KUKA KRL program: MyProgram_182().src

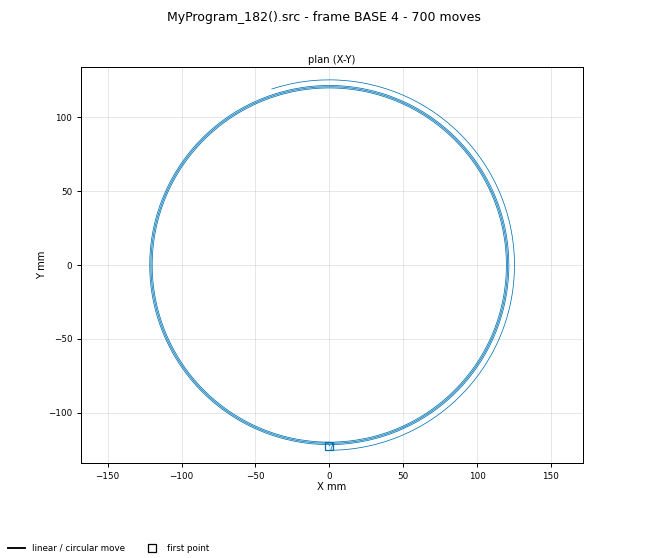
[picture p0: tool path of MyProgram_182().src in frame BASE 4, 700 of 700 moves have a stored position in this frame; points joined in program order, loops and branches not executed]
&ACCESS RVP
&REL 1
&PARAM TEMPLATE = C:\KRC\Roboter\Template\vorgabe
&PARAM EDITMASK = *
DEF MyProgram_182()
; ---- Setting reference (Base) ----
$BASE = BASE_DATA[4]

; --------------------------
; ---- Setting tool (TCP) ----
$TOOL = TOOL_DATA[3]
; --------------------------

$VEL.CP = VEL_APROX_PRINT
Startdeposition()
$VEL.CP = VEL_PRINT
LIN {X -0.1714,Y -122.3614,Z 133,A -93.0303,B 24.9608,C -1.4469,E1 25.0014,E2 179.2424} C_DIS
Enddeposition()
LIN {X 0.8695,Y -121.5175,Z 133,A -93.1539,B 24.9616,C -1.4326,E1 25.001,E2 179.3998} C_DIS
Startdeposition()
$VEL.CP = VEL_PRINT
LIN {X -1.6199,Y -121.5128,Z 133,A -95.084,B 24.9634,C -1.3971,E1 24.9954,E2 181.4142} C_DIS
LIN {X -5.9089,Y -121.3798,Z 133,A -96.2452,B 24.9613,C -1.437,E1 24.9924,E2 182.4809} C_DIS
LIN {X -12.044,Y -120.9259,Z 133,A -99.4115,B 24.962,C -1.4246,E1 24.9835,E2 185.6781} C_DIS
LIN {X -17.4797,Y -120.2602,Z 133,A -101.7782,B 24.9614,C -1.435,E1 24.977,E2 188.0216} C_DIS
LIN {X -21.0401,Y -119.6879,Z 133,A -103.7397,B 24.962,C -1.4234,E1 24.9715,E2 190.0125} C_DIS
LIN {X -24.264,Y -119.0756,Z 133,A -105.5719,B 24.9627,C -1.411,E1 24.9664,E2 191.8764} C_DIS
LIN {X -29.5809,Y -117.8675,Z 133,A -107.8497,B 24.9619,C -1.4258,E1 24.9603,E2 194.1221} C_DIS
LIN {X -32.4256,Y -117.1176,Z 133,A -109.326,B 24.9621,C -1.4225,E1 24.9563,E2 195.6083} C_DIS
LIN {X -36.1039,Y -116.0375,Z 133,A -111.1589,B 24.9621,C -1.4227,E1 24.9514,E2 197.444} C_DIS
LIN {X -40.6433,Y -114.5267,Z 133,A -113.43,B 24.9621,C -1.4239,E1 24.9454,E2 199.7166} C_DIS
LIN {X -44.0347,Y -113.2641,Z 133,A -115.0276,B 24.9617,C -1.4305,E1 24.9412,E2 201.3019} C_DIS
LIN {X -49.4851,Y -110.9909,Z 133,A -117.8563,B 24.9617,C -1.4314,E1 24.934,E2 204.1348} C_DIS
LIN {X -52.5926,Y -109.5528,Z 133,A -119.7843,B 24.9623,C -1.4192,E1 24.929,E2 206.0968} C_DIS
LIN {X -55.6549,Y -108.031,Z 133,A -121.1723,B 24.9616,C -1.4313,E1 24.9256,E2 207.4598} C_DIS
LIN {X -59.6628,Y -105.8704,Z 133,A -123.3001,B 24.9614,C -1.4352,E1 24.9204,E2 209.5846} C_DIS
LIN {X -62.5934,Y -104.165,Z 133,A -125.1136,B 24.9618,C -1.4279,E1 24.916,E2 211.4209} C_DIS
LIN {X -66.9605,Y -101.4123,Z 133,A -127.3139,B 24.961,C -1.4422,E1 24.9109,E2 213.5943} C_DIS
LIN {X -72.1767,Y -97.7684,Z 133,A -130.3221,B 24.9608,C -1.4469,E1 24.9041,E2 216.6016} C_DIS
LIN {X -75.3691,Y -95.3299,Z 133,A -132.2793,B 24.9608,C -1.4476,E1 24.8998,E2 218.5644} C_DIS
LIN {X -78.4994,Y -92.7685,Z 133,A -134.1769,B 24.9605,C -1.4517,E1 24.8957,E2 220.4595} C_DIS
LIN {X -81.6362,Y -90.0204,Z 133,A -135.8524,B 24.9596,C -1.4685,E1 24.8923,E2 222.1017} C_DIS
LIN {X -84.8955,Y -86.9542,Z 133,A -138.4312,B 24.9605,C -1.4522,E1 24.887,E2 224.7299} C_DIS
LIN {X -88.5295,Y -83.2516,Z 133,A -140.5025,B 24.9593,C -1.4741,E1 24.883,E2 226.7581} C_DIS
LIN {X -90.7073,Y -80.8729,Z 133,A -142.282,B 24.9597,C -1.4661,E1 24.8796,E2 228.5643} C_DIS
LIN {X -93.9091,Y -77.1324,Z 133,A -144.7365,B 24.9597,C -1.4658,E1 24.8752,E2 231.0309} C_DIS
LIN {X -96.8725,Y -73.375,Z 133,A -146.936,B 24.9593,C -1.4738,E1 24.8715,E2 233.2217} C_DIS
LIN {X -99.5155,Y -69.7483,Z 133,A -148.943,B 24.9587,C -1.4839,E1 24.8682,E2 235.2145} C_DIS
LIN {X -101.2493,Y -67.2069,Z 133,A -150.5671,B 24.959,C -1.4802,E1 24.8657,E2 236.8557} C_DIS
LIN {X -103.6846,Y -63.3844,Z 133,A -152.5823,B 24.9583,C -1.4911,E1 24.8627,E2 238.8551} C_DIS
LIN {X -105.425,Y -60.4464,Z 133,A -154.7129,B 24.9593,C -1.4731,E1 24.8597,E2 241.0398} C_DIS
LIN {X -107.529,Y -56.6154,Z 133,A -156.1389,B 24.9575,C -1.5062,E1 24.8579,E2 242.3945} C_DIS
LIN {X -109.0325,Y -53.6618,Z 133,A -157.753,B 24.9574,C -1.5083,E1 24.8559,E2 244.0121} C_DIS
LIN {X -110.2041,Y -51.2135,Z 133,A -159.1619,B 24.9574,C -1.5064,E1 24.8542,E2 245.4333} C_DIS
LIN {X -112.0151,Y -47.1208,Z 133,A -161.1145,B 24.9568,C -1.5194,E1 24.852,E2 247.3658} C_DIS
LIN {X -113.0996,Y -44.4581,Z 133,A -162.6444,B 24.957,C -1.5159,E1 24.8504,E2 248.9126} C_DIS
LIN {X -114.5797,Y -40.4958,Z 133,A -165.1319,B 24.9578,C -1.5007,E1 24.8481,E2 251.4502} C_DIS
LIN {X -115.9774,Y -36.2992,Z 133,A -166.7405,B 24.9563,C -1.5274,E1 24.8467,E2 253.0044} C_DIS
LIN {X -117.0095,Y -32.8111,Z 133,A -168.3362,B 24.9557,C -1.5379,E1 24.8455,E2 254.5845} C_DIS
LIN {X -117.8307,Y -29.726,Z 133,A -169.9109,B 24.9556,C -1.5396,E1 24.8444,E2 256.1642} C_DIS
LIN {X -118.7261,Y -25.9215,Z 133,A -171.7761,B 24.9553,C -1.5444,E1 24.8432,E2 258.0289} C_DIS
LIN {X -119.4847,Y -22.1777,Z 133,A -173.7085,B 24.9553,C -1.5444,E1 24.8422,E2 259.9726} C_DIS
LIN {X -120.082,Y -18.6588,Z 133,A -175.2045,B 24.9545,C -1.5579,E1 24.8416,E2 261.4455} C_DIS
LIN {X -120.5511,Y -15.3426,Z 133,A -177.0022,B 24.9548,C -1.5536,E1 24.8409,E2 263.2642} C_DIS
LIN {X -121.1464,Y -9.5742,Z 133,A -179.7063,B 24.9542,C -1.5637,E1 24.8402,E2 265.9603} C_DIS
LIN {X -121.3814,Y -5.8756,Z 133,A 178.598,B 24.9537,C -1.5716,E1 24.8399,E2 267.6474} C_DIS
LIN {X -121.5254,Y 0.0221,Z 133,A 175.7482,B 24.9534,C -1.5778,E1 24.8398,E2 270.4998} C_DIS
LIN {X -121.3885,Y 5.7327,Z 133,A 173.2315,B 24.9524,C -1.5941,E1 24.84,E2 272.9926} C_DIS
LIN {X -121.191,Y 8.9707,Z 133,A 171.3253,B 24.953,C -1.5832,E1 24.8404,E2 274.9364} C_DIS
LIN {X -120.7228,Y 13.9263,Z 133,A 169.1754,B 24.9521,C -1.5992,E1 24.841,E2 277.061} C_DIS
LIN {X -120.2359,Y 17.6498,Z 133,A 167.4666,B 24.9516,C -1.6076,E1 24.8416,E2 278.7599} C_DIS
LIN {X -119.6712,Y 21.1333,Z 133,A 165.9207,B 24.9509,C -1.6181,E1 24.8423,E2 280.2901} C_DIS
LIN {X -119.212,Y 23.5938,Z 133,A 164.3598,B 24.9517,C -1.6057,E1 24.8432,E2 281.8898} C_DIS
LIN {X -118.2189,Y 28.1465,Z 133,A 162.2925,B 24.9509,C -1.6183,E1 24.8445,E2 283.9391} C_DIS
LIN {X -117.2416,Y 31.9811,Z 133,A 160.3797,B 24.9507,C -1.6223,E1 24.8458,E2 285.8536} C_DIS
LIN {X -116.311,Y 35.2093,Z 133,A 158.6706,B 24.9507,C -1.622,E1 24.8472,E2 287.5731} C_DIS
LIN {X -114.606,Y 40.4198,Z 133,A 156.1475,B 24.95,C -1.6328,E1 24.8495,E2 290.0849} C_DIS
LIN {X -113.2622,Y 44.0395,Z 133,A 154.6517,B 24.9488,C -1.6524,E1 24.8509,E2 291.5424} C_DIS
LIN {X -111.9631,Y 47.2453,Z 133,A 152.7073,B 24.9494,C -1.6441,E1 24.853,E2 293.5175} C_DIS
LIN {X -110.3469,Y 50.9041,Z 133,A 150.9642,B 24.9486,C -1.656,E1 24.855,E2 295.2419} C_DIS
LIN {X -109.2384,Y 53.245,Z 133,A 149.0187,B 24.9503,C -1.6289,E1 24.8575,E2 297.2624} C_DIS
LIN {X -107.0191,Y 57.5774,Z 133,A 146.7211,B 24.9499,C -1.6356,E1 24.8605,E2 299.5562} C_DIS
LIN {X -104.6811,Y 61.7255,Z 133,A 145.3326,B 24.9472,C -1.6786,E1 24.8623,E2 300.8493} C_DIS
LIN {X -100.2308,Y 68.7165,Z 133,A 141.1386,B 24.9472,C -1.6774,E1 24.8687,E2 305.0674} C_DIS
LIN {X -97.9703,Y 71.9019,Z 133,A 139.3158,B 24.9469,C -1.6833,E1 24.8716,E2 306.8851} C_DIS
LIN {X -95.4946,Y 75.1596,Z 133,A 137.3071,B 24.9468,C -1.6851,E1 24.8751,E2 308.8989} C_DIS
LIN {X -92.8236,Y 78.4345,Z 133,A 135.3193,B 24.9464,C -1.6906,E1 24.8786,E2 310.8829} C_DIS
LIN {X -90.3001,Y 81.3277,Z 133,A 133.4255,B 24.9464,C -1.6916,E1 24.8821,E2 312.7827} C_DIS
LIN {X -87.1093,Y 84.7363,Z 133,A 131.2611,B 24.9459,C -1.6988,E1 24.8863,E2 314.9396} C_DIS
LIN {X -84.2652,Y 87.5645,Z 133,A 129.3791,B 24.9456,C -1.7037,E1 24.89,E2 316.8175} C_DIS
LIN {X -81.1545,Y 90.4552,Z 133,A 127.342,B 24.9454,C -1.7069,E1 24.8942,E2 318.8552} C_DIS
LIN {X -77.9713,Y 93.2126,Z 133,A 125.4465,B 24.9449,C -1.7154,E1 24.8982,E2 320.738} C_DIS
LIN {X -74.8032,Y 95.7746,Z 133,A 123.3839,B 24.9449,C -1.7134,E1 24.9028,E2 322.813} C_DIS
LIN {X -71.0844,Y 98.5665,Z 133,A 121.1715,B 24.9447,C -1.7171,E1 24.9077,E2 325.0243} C_DIS
LIN {X -67.5256,Y 101.0364,Z 133,A 119.4573,B 24.9435,C -1.7356,E1 24.9116,E2 326.7003} C_DIS
LIN {X -64.1253,Y 103.2284,Z 133,A 117.0152,B 24.9448,C -1.7159,E1 24.9175,E2 329.1971} C_DIS
LIN {X -61.3323,Y 104.9117,Z 133,A 115.7211,B 24.944,C -1.7293,E1 24.9205,E2 330.4632} C_DIS
LIN {X -57.7529,Y 106.9251,Z 133,A 113.5487,B 24.9444,C -1.7223,E1 24.9259,E2 332.6585} C_DIS
LIN {X -53.5846,Y 109.0707,Z 133,A 111.6337,B 24.9433,C -1.739,E1 24.9306,E2 334.5389} C_DIS
LIN {X -49.7713,Y 110.8628,Z 133,A 109.6684,B 24.9431,C -1.743,E1 24.9356,E2 336.4995} C_DIS
LIN {X -47.024,Y 112.0556,Z 133,A 108.269,B 24.9429,C -1.7457,E1 24.9392,E2 337.8959} C_DIS
LIN {X -41.3309,Y 114.2785,Z 133,A 105.3623,B 24.9427,C -1.7484,E1 24.9468,E2 340.8022} C_DIS
LIN {X -38.0593,Y 115.4093,Z 133,A 103.6121,B 24.9429,C -1.7452,E1 24.9514,E2 342.5634} C_DIS
LIN {X -33.9229,Y 116.6918,Z 133,A 101.5952,B 24.9427,C -1.7486,E1 24.9568,E2 344.5756} C_DIS
LIN {X -30.0844,Y 117.7399,Z 133,A 99.7639,B 24.9424,C -1.7525,E1 24.9617,E2 346.4004} C_DIS
LIN {X -27.4403,Y 118.3855,Z 133,A 98.1282,B 24.9434,C -1.7379,E1 24.9663,E2 348.0729} C_DIS
LIN {X -24.2011,Y 119.0884,Z 133,A 97.0595,B 24.9418,C -1.7614,E1 24.969,E2 349.087} C_DIS
LIN {X -18.4586,Y 120.113,Z 133,A 94.1674,B 24.9421,C -1.7571,E1 24.977,E2 351.9923} C_DIS
LIN {X -15.4534,Y 120.5366,Z 133,A 91.9287,B 24.9444,C -1.7217,E1 24.9835,E2 354.3165} C_DIS
LIN {X -9.9847,Y 121.1119,Z 133,A 90.4873,B 24.941,C -1.7749,E1 24.9871,E2 355.6325} C_DIS
LIN {X -4.1146,Y 121.4544,Z 133,A 87.4557,B 24.9417,C -1.764,E1 24.9957,E2 358.6908} C_DIS
LIN {X 2.7806,Y 121.4924,Z 133,A 83.7604,B 24.943,C -1.7443,E1 25.0061,E2 362.4325} C_DIS
LIN {X 6.1114,Y 121.3697,Z 133,A 82.3946,B 24.9424,C -1.7538,E1 25.0098,E2 363.7754} C_DIS
LIN {X 9.304,Y 121.1666,Z 133,A 80.4497,B 24.9437,C -1.7338,E1 25.0154,E2 365.7668} C_DIS
LIN {X 13.7722,Y 120.7407,Z 133,A 78.9161,B 24.9419,C -1.7601,E1 25.0195,E2 367.237} C_DIS
LIN {X 17.8606,Y 120.2057,Z 133,A 76.8319,B 24.9424,C -1.7531,E1 25.0253,E2 369.336} C_DIS
LIN {X 21.3951,Y 119.6246,Z 133,A 75.0487,B 24.9427,C -1.7482,E1 25.0302,E2 371.129} C_DIS
LIN {X 26.4333,Y 118.6147,Z 133,A 72.8052,B 24.9423,C -1.7552,E1 25.0363,E2 373.3528} C_DIS
LIN {X 30.0915,Y 117.7381,Z 133,A 71.1132,B 24.9421,C -1.758,E1 25.0408,E2 375.0358} C_DIS
LIN {X 33.5438,Y 116.8029,Z 133,A 69.4281,B 24.9421,C -1.7569,E1 25.0454,E2 376.7208} C_DIS
LIN {X 37.679,Y 115.5357,Z 133,A 67.2523,B 24.9427,C -1.7489,E1 25.0512,E2 378.9115} C_DIS
LIN {X 40.9856,Y 114.4031,Z 133,A 65.7299,B 24.9424,C -1.7533,E1 25.0552,E2 380.4204} C_DIS
LIN {X 47.3838,Y 111.9053,Z 133,A 62.4044,B 24.9429,C -1.7458,E1 25.0638,E2 383.7561} C_DIS
LIN {X 52.9272,Y 109.3927,Z 133,A 59.5132,B 24.9432,C -1.7414,E1 25.0712,E2 386.6505} C_DIS
LIN {X 56.3187,Y 107.6851,Z 133,A 57.82,B 24.943,C -1.7436,E1 25.0754,E2 388.3338} C_DIS
LIN {X 59.7529,Y 105.8199,Z 133,A 55.319,B 24.9452,C -1.7099,E1 25.0816,E2 390.907} C_DIS
LIN {X 64.0474,Y 103.2768,Z 133,A 53.7251,B 24.9431,C -1.7422,E1 25.0852,E2 392.4197} C_DIS
LIN {X 69.0589,Y 99.9957,Z 133,A 50.7198,B 24.944,C -1.7289,E1 25.0923,E2 395.4464} C_DIS
LIN {X 72.9607,Y 97.1859,Z 133,A 48.6037,B 24.9438,C -1.7321,E1 25.097,E2 397.5474} C_DIS
LIN {X 75.8072,Y 94.9809,Z 133,A 46.8061,B 24.9443,C -1.7241,E1 25.101,E2 399.3572} C_DIS
LIN {X 79.2112,Y 92.1619,Z 133,A 44.7655,B 24.9444,C -1.7221,E1 25.1053,E2 401.3946} C_DIS
LIN {X 82.2523,Y 89.4574,Z 133,A 43.1469,B 24.9437,C -1.7327,E1 25.1086,E2 402.9817} C_DIS
LIN {X 85.4415,Y 86.4173,Z 133,A 40.7559,B 24.945,C -1.7131,E1 25.1135,E2 405.4091} C_DIS
LIN {X 88.7384,Y 83.0292,Z 133,A 38.49,B 24.9454,C -1.7063,E1 25.1179,E2 407.6811} C_DIS
LIN {X 91.8422,Y 79.5817,Z 133,A 36.4182,B 24.9454,C -1.7068,E1 25.1217,E2 409.7424} C_DIS
LIN {X 95.331,Y 75.3678,Z 133,A 33.7885,B 24.946,C -1.6982,E1 25.1263,E2 412.3805} C_DIS
LIN {X 97.7085,Y 72.2582,Z 133,A 31.9897,B 24.9461,C -1.6958,E1 25.1294,E2 414.1761} C_DIS
LIN {X 101.2183,Y 67.2533,Z 133,A 29.0556,B 24.9467,C -1.6859,E1 25.134,E2 417.1193} C_DIS
LIN {X 103.1728,Y 64.215,Z 133,A 27.6255,B 24.9462,C -1.6947,E1 25.1361,E2 418.5213} C_DIS
LIN {X 105.044,Y 61.1053,Z 133,A 25.7489,B 24.947,C -1.6819,E1 25.1388,E2 420.4184} C_DIS
LIN {X 107.0074,Y 57.5991,Z 133,A 23.8134,B 24.9474,C -1.6747,E1 25.1414,E2 422.361} C_DIS
LIN {X 109.006,Y 53.7155,Z 133,A 21.2767,B 24.9493,C -1.6455,E1 25.1447,E2 424.9529} C_DIS
LIN {X 110.9245,Y 49.6335,Z 133,A 19.6987,B 24.948,C -1.6662,E1 25.1464,E2 426.4735} C_DIS
LIN {X 112.5458,Y 45.8395,Z 133,A 17.6274,B 24.9487,C -1.6543,E1 25.1487,E2 428.5616} C_DIS
LIN {X 114.2892,Y 41.3014,Z 133,A 15.5706,B 24.9484,C -1.659,E1 25.1506,E2 430.5957} C_DIS
LIN {X 115.4115,Y 38.0527,Z 133,A 13.8382,B 24.9491,C -1.6486,E1 25.1522,E2 432.343} C_DIS
LIN {X 116.909,Y 33.1693,Z 133,A 11.4999,B 24.9493,C -1.6446,E1 25.1541,E2 434.6773} C_DIS
LIN {X 117.9396,Y 29.2965,Z 133,A 9.2966,B 24.9506,C -1.6232,E1 25.1556,E2 436.9183} C_DIS
LIN {X 118.7103,Y 25.9949,Z 133,A 7.7401,B 24.9508,C -1.6202,E1 25.1565,E2 438.4728} C_DIS
LIN {X 119.3724,Y 22.7623,Z 133,A 6.0818,B 24.9514,C -1.6102,E1 25.1574,E2 440.1449} C_DIS
LIN {X 120.032,Y 18.9807,Z 133,A 3.7513,B 24.9533,C -1.5789,E1 25.1584,E2 442.5357} C_DIS
LIN {X 120.8602,Y 12.6811,Z 133,A 1.024,B 24.9531,C -1.5823,E1 25.1592,E2 445.2387} C_DIS
LIN {X 121.2876,Y 7.5595,Z 133,A -0.6208,B 24.9513,C -1.6129,E1 25.1595,E2 446.8016} C_DIS
LIN {X 121.5233,Y 0.4226,Z 133,A -3.7776,B 24.9513,C -1.6123,E1 25.1598,E2 449.941} C_DIS
LIN {X 121.5038,Y -2.1482,Z 133,A -5.3004,B 24.9525,C -1.5928,E1 25.1598,E2 451.5006} C_DIS
LIN {X 121.3612,Y -6.2818,Z 133,A -7.1686,B 24.9526,C -1.5905,E1 25.1595,E2 453.3633} C_DIS
LIN {X 121.0842,Y -10.3146,Z 133,A -8.9077,B 24.9525,C -1.5926,E1 25.1592,E2 455.0872} C_DIS
LIN {X 120.1422,Y -18.2707,Z 133,A -12.5694,B 24.9529,C -1.5859,E1 25.1579,E2 458.743} C_DIS
LIN {X 119.0748,Y -24.2677,Z 133,A -15.5726,B 24.9538,C -1.5699,E1 25.1564,E2 461.7664} C_DIS
LIN {X 117.9952,Y -29.0716,Z 133,A -18.0282,B 24.9547,C -1.5556,E1 25.1548,E2 464.2413} C_DIS
LIN {X 117.0701,Y -32.595,Z 133,A -19.6657,B 24.9547,C -1.5541,E1 25.1536,E2 465.8729} C_DIS
LIN {X 114.9989,Y -39.2852,Z 133,A -22.999,B 24.9555,C -1.542,E1 25.1508,E2 469.216} C_DIS
LIN {X 113.7527,Y -42.7553,Z 133,A -24.6508,B 24.9555,C -1.5408,E1 25.1492,E2 470.8612} C_DIS
LIN {X 112.8471,Y -45.0941,Z 133,A -26.4568,B 24.9575,C -1.5062,E1 25.1473,E2 472.7388} C_DIS
LIN {X 111.0301,Y -49.3975,Z 133,A -28.0517,B 24.9562,C -1.5294,E1 25.1456,E2 474.2703} C_DIS
LIN {X 109.6975,Y -52.2901,Z 133,A -29.4513,B 24.9562,C -1.5299,E1 25.1439,E2 475.6612} C_DIS
LIN {X 108.5654,Y -54.6031,Z 133,A -31.582,B 24.9589,C -1.481,E1 25.1411,E2 477.8959} C_DIS
LIN {X 105.7915,Y -59.8034,Z 133,A -33.5921,B 24.9573,C -1.5105,E1 25.1385,E2 479.826} C_DIS
LIN {X 103.7664,Y -63.2509,Z 133,A -35.4123,B 24.9573,C -1.5082,E1 25.1359,E2 481.6423} C_DIS
LIN {X 101.6599,Y -66.5854,Z 133,A -37.3409,B 24.9579,C -1.4994,E1 25.1329,E2 483.5819} C_DIS
LIN {X 99.1324,Y -70.2919,Z 133,A -39.3276,B 24.9579,C -1.4998,E1 25.1298,E2 485.5579} C_DIS
LIN {X 97.0862,Y -73.0925,Z 133,A -41.3737,B 24.9592,C -1.475,E1 25.1263,E2 487.6527} C_DIS
LIN {X 94.7461,Y -76.1005,Z 133,A -42.7678,B 24.9584,C -1.49,E1 25.1239,E2 489.005} C_DIS
LIN {X 92.1415,Y -79.2349,Z 133,A -44.5126,B 24.9582,C -1.4936,E1 25.1208,E2 490.7333} C_DIS
LIN {X 89.5008,Y -82.205,Z 133,A -46.9333,B 24.96,C -1.4619,E1 25.1162,E2 493.2181} C_DIS
LIN {X 86.835,Y -85.0169,Z 133,A -48.3815,B 24.9592,C -1.4758,E1 25.1134,E2 494.6271} C_DIS
LIN {X 83.9149,Y -87.8997,Z 133,A -49.9871,B 24.9586,C -1.4873,E1 25.1103,E2 496.1989} C_DIS
LIN {X 80.9349,Y -90.6517,Z 133,A -52.4468,B 24.9603,C -1.4559,E1 25.1051,E2 498.7229} C_DIS
LIN {X 78.5169,Y -92.7537,Z 133,A -53.7327,B 24.9599,C -1.4634,E1 25.1024,E2 499.9861} C_DIS
LIN {X 75.1717,Y -95.485,Z 133,A -55.677,B 24.9599,C -1.4634,E1 25.0982,E2 501.9233} C_DIS
LIN {X 71.5873,Y -98.2009,Z 133,A -57.8821,B 24.9604,C -1.4546,E1 25.0932,E2 504.1409} C_DIS
LIN {X 68.4742,Y -100.3971,Z 133,A -59.6699,B 24.9605,C -1.4513,E1 25.0891,E2 505.9304} C_DIS
LIN {X 64.6916,Y -102.8752,Z 133,A -61.7482,B 24.9606,C -1.4498,E1 25.0842,E2 508.0057} C_DIS
LIN {X 61.9595,Y -104.5431,Z 133,A -63.6503,B 24.9618,C -1.4279,E1 25.0796,E2 509.9535} C_DIS
LIN {X 58.5648,Y -106.4817,Z 133,A -65.0836,B 24.9609,C -1.4444,E1 25.0762,E2 511.3437} C_DIS
LIN {X 55.3771,Y -108.1722,Z 133,A -66.8756,B 24.9613,C -1.4371,E1 25.0717,E2 513.1479} C_DIS
LIN {X 47.1492,Y -112.0033,Z 133,A -71.9012,B 24.9636,C -1.3949,E1 25.0586,E2 518.2609} C_DIS
LIN {X 41.4943,Y -114.2195,Z 133,A -73.8492,B 24.9614,C -1.4345,E1 25.0538,E2 520.111} C_DIS
LIN {X 38.1565,Y -115.3769,Z 133,A -75.5105,B 24.9616,C -1.4326,E1 25.0494,E2 521.7736} C_DIS
LIN {X 34.508,Y -116.5204,Z 133,A -77.4906,B 24.9621,C -1.4221,E1 25.0441,E2 523.7752} C_DIS
LIN {X 28.9212,Y -118.0316,Z 133,A -80.0191,B 24.9618,C -1.4287,E1 25.0373,E2 526.2841} C_DIS
LIN {X 25.7525,Y -118.7626,Z 133,A -82.4347,B 24.964,C -1.3857,E1 25.0304,E2 528.7984} C_DIS
LIN {X 19.9721,Y -119.87,Z 133,A -84.4325,B 24.9622,C -1.42,E1 25.0251,E2 530.7128} C_DIS
LIN {X 12.8123,Y -120.846,Z 133,A -87.5006,B 24.9615,C -1.4337,E1 25.0168,E2 533.7459} C_DIS
LIN {X 7.3926,Y -121.298,Z 133,A -90.2146,B 24.9619,C -1.4254,E1 25.0092,E2 536.4783} C_DIS
LIN {X 1.4948,Y -121.515,Z 133,A -93.1207,B 24.9623,C -1.4186,E1 25.001,E2 539.3998} C_DIS
LIN {X 1.4948,Y -121.515,Z 133,A -93.1207,B 24.9623,C -1.4186,E1 25.001,E2 539.3998} C_DIS
Enddeposition()
LIN {X 0.8662,Y -120.6827,Z 133,A -93.1944,B 24.961,C -1.4437,E1 25.001,E2 539.414} C_DIS
Startdeposition()
$VEL.CP = VEL_PRINT
LIN {X 6.735,Y -120.5001,Z 133,A -89.6486,B 24.959,C -1.4803,E1 25.0111,E2 535.7825} C_DIS
LIN {X 11.2298,Y -120.1633,Z 133,A -87.692,B 24.9594,C -1.4727,E1 25.0165,E2 533.8449} C_DIS
LIN {X 15.1137,Y -119.7371,Z 133,A -85.2133,B 24.9576,C -1.5037,E1 25.0235,E2 531.2947} C_DIS
LIN {X 19.8381,Y -119.044,Z 133,A -83.9162,B 24.9601,C -1.459,E1 25.0268,E2 530.1047} C_DIS
LIN {X 22.402,Y -118.5895,Z 133,A -82.1059,B 24.9586,C -1.4874,E1 25.032,E2 528.2293} C_DIS
LIN {X 25.9487,Y -117.8641,Z 133,A -80.5996,B 24.959,C -1.4787,E1 25.036,E2 526.7453} C_DIS
LIN {X 29.8463,Y -116.9369,Z 133,A -78.7947,B 24.9592,C -1.476,E1 25.0409,E2 524.9495} C_DIS
LIN {X 34.6476,Y -115.6074,Z 133,A -76.5132,B 24.9592,C -1.4746,E1 25.047,E2 522.6752} C_DIS
LIN {X 38.4892,Y -114.3839,Z 133,A -74.6164,B 24.9592,C -1.4762,E1 25.052,E2 520.7782} C_DIS
LIN {X 41.1746,Y -113.4452,Z 133,A -73.231,B 24.959,C -1.4796,E1 25.0557,E2 519.3876} C_DIS
LIN {X 45.3095,Y -111.8575,Z 133,A -71.0621,B 24.9586,C -1.4858,E1 25.0614,E2 517.2088} C_DIS
LIN {X 48.3168,Y -110.5929,Z 133,A -69.5419,B 24.9586,C -1.4867,E1 25.0653,E2 515.6901} C_DIS
LIN {X 51.3605,Y -109.2141,Z 133,A -67.3897,B 24.9569,C -1.5168,E1 25.0709,E2 513.4722} C_DIS
LIN {X 55.1226,Y -107.3628,Z 133,A -65.8728,B 24.958,C -1.497,E1 25.0745,E2 512.0063} C_DIS
LIN {X 58.9565,Y -105.307,Z 133,A -63.7704,B 24.9577,C -1.5025,E1 25.0797,E2 509.8971} C_DIS
LIN {X 62.6065,Y -103.1787,Z 133,A -61.9393,B 24.958,C -1.4977,E1 25.084,E2 508.0829} C_DIS
LIN {X 65.7074,Y -101.2326,Z 133,A -60.166,B 24.9577,C -1.5028,E1 25.0882,E2 506.3032} C_DIS
LIN {X 68.7385,Y -99.1995,Z 133,A -58.3841,B 24.9574,C -1.5088,E1 25.0924,E2 504.5133} C_DIS
LIN {X 71.4896,Y -97.2348,Z 133,A -56.7625,B 24.9571,C -1.513,E1 25.096,E2 502.8875} C_DIS
LIN {X 74.793,Y -94.7183,Z 133,A -54.8043,B 24.9569,C -1.5167,E1 25.1003,E2 500.9278} C_DIS
LIN {X 78.0511,Y -92.0514,Z 133,A -52.8709,B 24.9569,C -1.518,E1 25.1045,E2 498.9988} C_DIS
LIN {X 81.0703,Y -89.4039,Z 133,A -51.0126,B 24.9567,C -1.5201,E1 25.1084,E2 497.1429} C_DIS
LIN {X 83.1894,Y -87.4356,Z 133,A -49.5486,B 24.9563,C -1.5279,E1 25.1114,E2 495.6665} C_DIS
LIN {X 86.3245,Y -84.3424,Z 133,A -47.4224,B 24.9559,C -1.5348,E1 25.1156,E2 493.5329} C_DIS
LIN {X 89.4784,Y -80.9884,Z 133,A -45.4147,B 24.9561,C -1.5316,E1 25.1193,E2 491.5416} C_DIS
LIN {X 91.198,Y -79.0472,Z 133,A -44.086,B 24.9556,C -1.5397,E1 25.1218,E2 490.1999} C_DIS
LIN {X 93.6544,Y -76.1208,Z 133,A -42.2334,B 24.9552,C -1.5465,E1 25.1251,E2 488.3399} C_DIS
LIN {X 96.3839,Y -72.6338,Z 133,A -40.1915,B 24.955,C -1.5492,E1 25.1286,E2 486.3012} C_DIS
LIN {X 98.6551,Y -69.5165,Z 133,A -38.3587,B 24.9547,C -1.5544,E1 25.1315,E2 484.4649} C_DIS
LIN {X 101.1563,Y -65.8252,Z 133,A -36.3286,B 24.9547,C -1.5561,E1 25.1347,E2 482.4409} C_DIS
LIN {X 103.1705,Y -62.62,Z 133,A -34.4579,B 24.9541,C -1.565,E1 25.1374,E2 480.5587} C_DIS
LIN {X 105.2736,Y -59.0161,Z 133,A -32.2728,B 24.9532,C -1.5811,E1 25.1405,E2 478.347} C_DIS
LIN {X 107.1627,Y -55.5145,Z 133,A -30.5832,B 24.9534,C -1.5768,E1 25.1427,E2 476.6766} C_DIS
LIN {X 108.8825,Y -52.0547,Z 133,A -28.8508,B 24.9534,C -1.5773,E1 25.1448,E2 474.9522} C_DIS
LIN {X 110.3252,Y -48.9239,Z 133,A -27.2403,B 24.9532,C -1.581,E1 25.1466,E2 473.3416} C_DIS
LIN {X 112.3237,Y -44.1443,Z 133,A -24.7257,B 24.9525,C -1.5915,E1 25.1493,E2 470.8164} C_DIS
LIN {X 113.7104,Y -40.4399,Z 133,A -22.8411,B 24.9522,C -1.5977,E1 25.1511,E2 468.9276} C_DIS
LIN {X 115.2244,Y -35.9012,Z 133,A -20.7712,B 24.9523,C -1.5948,E1 25.1529,E2 466.8761} C_DIS
LIN {X 116.4661,Y -31.641,Z 133,A -18.5058,B 24.9515,C -1.6096,E1 25.1546,E2 464.589} C_DIS
LIN {X 117.4701,Y -27.6819,Z 133,A -16.6291,B 24.9513,C -1.6127,E1 25.1558,E2 462.7157} C_DIS
LIN {X 118.0669,Y -25.0091,Z 133,A -15.3358,B 24.951,C -1.6166,E1 25.1566,E2 461.4207} C_DIS
LIN {X 119.003,Y -20.0836,Z 133,A -12.9704,B 24.9506,C -1.6237,E1 25.1578,E2 459.0526} C_DIS
LIN {X 119.6083,Y -16.097,Z 133,A -11.0405,B 24.9502,C -1.6307,E1 25.1585,E2 457.1175} C_DIS
LIN {X 120.0406,Y -12.4766,Z 133,A -9.1741,B 24.9494,C -1.6432,E1 25.1591,E2 455.2328} C_DIS
LIN {X 120.3587,Y -8.8781,Z 133,A -7.7037,B 24.9498,C -1.6365,E1 25.1594,E2 453.7867} C_DIS
LIN {X 120.5813,Y -5.0419,Z 133,A -5.3533,B 24.9478,C -1.669,E1 25.1597,E2 451.3738} C_DIS
LIN {X 120.6843,Y -0.8322,Z 133,A -4.0936,B 24.9497,C -1.6384,E1 25.1598,E2 450.1938} C_DIS
LIN {X 120.4929,Y 6.8561,Z 133,A -0.3562,B 24.9487,C -1.6545,E1 25.1595,E2 446.4406} C_DIS
LIN {X 120.0138,Y 12.7237,Z 133,A 2.4177,B 24.9482,C -1.6625,E1 25.1588,E2 443.6643} C_DIS
LIN {X 119.2875,Y 18.3212,Z 133,A 4.8833,B 24.9483,C -1.6604,E1 25.1579,E2 441.2181} C_DIS
LIN {X 118.8659,Y 20.8824,Z 133,A 6.4155,B 24.9472,C -1.6793,E1 25.1572,E2 439.6504} C_DIS
LIN {X 117.6649,Y 26.8355,Z 133,A 9.271,B 24.9467,C -1.687,E1 25.1555,E2 436.7934} C_DIS
LIN {X 116.8142,Y 30.3303,Z 133,A 10.8697,B 24.9467,C -1.6869,E1 25.1544,E2 435.2042} C_DIS
LIN {X 116.0155,Y 33.2549,Z 133,A 12.5224,B 24.9457,C -1.702,E1 25.1532,E2 433.5253} C_DIS
LIN {X 114.9539,Y 36.7524,Z 133,A 14.1257,B 24.9457,C -1.7007,E1 25.1519,E2 431.9341} C_DIS
LIN {X 113.7344,Y 40.3735,Z 133,A 16.0713,B 24.945,C -1.7128,E1 25.1501,E2 429.9712} C_DIS
LIN {X 112.3052,Y 44.1921,Z 133,A 18.2857,B 24.9438,C -1.7324,E1 25.1478,E2 427.7226} C_DIS
LIN {X 110.8723,Y 47.6707,Z 133,A 19.3544,B 24.9457,C -1.702,E1 25.1467,E2 426.7314} C_DIS
LIN {X 108.2462,Y 53.3641,Z 133,A 22.2445,B 24.9454,C -1.7063,E1 25.1433,E2 423.8469} C_DIS
LIN {X 107.2837,Y 55.2784,Z 133,A 23.7221,B 24.9438,C -1.7318,E1 25.1414,E2 422.317} C_DIS
LIN {X 105.0646,Y 59.3887,Z 133,A 25.914,B 24.9435,C -1.7367,E1 25.1384,E2 420.125} C_DIS
LIN {X 102.292,Y 64.047,Z 133,A 28.4641,B 24.9431,C -1.7424,E1 25.1347,E2 417.5743} C_DIS
LIN {X 98.3866,Y 69.8972,Z 133,A 31.4241,B 24.9438,C -1.7324,E1 25.1302,E2 414.6526} C_DIS
LIN {X 96.9869,Y 71.8263,Z 133,A 32.8566,B 24.9426,C -1.75,E1 25.1277,E2 413.1854} C_DIS
LIN {X 94.5573,Y 74.9962,Z 133,A 34.7474,B 24.9423,C -1.7544,E1 25.1245,E2 411.2932} C_DIS
LIN {X 91.6852,Y 78.4827,Z 133,A 36.8643,B 24.9421,C -1.7582,E1 25.1207,E2 409.1772} C_DIS
LIN {X 89.1907,Y 81.3047,Z 133,A 38.6816,B 24.9417,C -1.7637,E1 25.1173,E2 407.3548} C_DIS
LIN {X 86.3065,Y 84.3608,Z 133,A 40.6272,B 24.9416,C -1.7658,E1 25.1135,E2 405.4128} C_DIS
LIN {X 83.2882,Y 87.3411,Z 133,A 42.374,B 24.9421,C -1.7571,E1 25.1101,E2 403.6937} C_DIS
LIN {X 81.0673,Y 89.4066,Z 133,A 44.0808,B 24.9411,C -1.773,E1 25.1065,E2 401.9563} C_DIS
LIN {X 78.0435,Y 92.0578,Z 133,A 45.9709,B 24.9409,C -1.7759,E1 25.1025,E2 400.0669} C_DIS
LIN {X 74.7798,Y 94.7287,Z 133,A 48.1165,B 24.9402,C -1.7866,E1 25.0978,E2 397.9039} C_DIS
LIN {X 70.9838,Y 97.605,Z 133,A 50.2551,B 24.9402,C -1.7847,E1 25.093,E2 395.7775} C_DIS
LIN {X 67.9,Y 99.7755,Z 133,A 52.1479,B 24.9398,C -1.7927,E1 25.0886,E2 393.8722} C_DIS
LIN {X 64.1851,Y 102.2054,Z 133,A 54.1158,B 24.94,C -1.7893,E1 25.084,E2 391.9187} C_DIS
LIN {X 61.198,Y 104.0203,Z 133,A 55.9266,B 24.9393,C -1.7991,E1 25.0796,E2 390.0904} C_DIS
LIN {X 57.7156,Y 105.9926,Z 133,A 57.703,B 24.9396,C -1.7959,E1 25.0753,E2 388.3268} C_DIS
LIN {X 54.1743,Y 107.8447,Z 133,A 59.5853,B 24.9394,C -1.7977,E1 25.0707,E2 386.4455} C_DIS
LIN {X 50.3236,Y 109.6932,Z 133,A 61.4015,B 24.9399,C -1.7901,E1 25.0661,E2 384.6518} C_DIS
LIN {X 47.9544,Y 110.7496,Z 133,A 62.7677,B 24.9394,C -1.7979,E1 25.0626,E2 383.2706} C_DIS
LIN {X 44.2939,Y 112.2657,Z 133,A 65.0352,B 24.938,C -1.8181,E1 25.0566,E2 380.9602} C_DIS
LIN {X 40.9642,Y 113.5212,Z 133,A 66.2577,B 24.9394,C -1.7976,E1 25.0535,E2 379.7888} C_DIS
LIN {X 37.7728,Y 114.6227,Z 133,A 68.0037,B 24.9389,C -1.8057,E1 25.0489,E2 378.027} C_DIS
LIN {X 33.6985,Y 115.8855,Z 133,A 69.8711,B 24.9393,C -1.7998,E1 25.0439,E2 376.1768} C_DIS
LIN {X 30.9478,Y 116.6508,Z 133,A 71.2612,B 24.9391,C -1.8024,E1 25.0402,E2 374.7829} C_DIS
LIN {X 27.4117,Y 117.5337,Z 133,A 72.9134,B 24.9393,C -1.7997,E1 25.0357,E2 373.1396} C_DIS
LIN {X 25.0788,Y 118.0519,Z 133,A 74.2035,B 24.9388,C -1.8075,E1 25.0321,E2 371.8324} C_DIS
LIN {X 21.318,Y 118.7883,Z 133,A 75.9638,B 24.9388,C -1.8055,E1 25.0273,E2 370.079} C_DIS
LIN {X 17.9129,Y 119.3508,Z 133,A 77.6938,B 24.9386,C -1.8103,E1 25.0225,E2 368.3394} C_DIS
LIN {X 14.0532,Y 119.8649,Z 133,A 79.4596,B 24.9388,C -1.8069,E1 25.0177,E2 366.5831} C_DIS
LIN {X 9.4842,Y 120.3142,Z 133,A 81.7092,B 24.9386,C -1.8103,E1 25.0114,E2 364.3266} C_DIS
LIN {X 5.6314,Y 120.5557,Z 133,A 83.8026,B 24.9378,C -1.8223,E1 25.0055,E2 362.2054} C_DIS
LIN {X 2.3577,Y 120.6632,Z 133,A 85.0216,B 24.9388,C -1.8066,E1 25.0022,E2 361.0239} C_DIS
LIN {X -3.9606,Y 120.6222,Z 133,A 87.9611,B 24.9391,C -1.8031,E1 24.994,E2 358.0926} C_DIS
LIN {X -9.5884,Y 120.3054,Z 133,A 90.9059,B 24.9383,C -1.8143,E1 24.9857,E2 355.1202} C_DIS
LIN {X -15.0638,Y 119.7437,Z 133,A 93.4,B 24.9388,C -1.8073,E1 24.9788,E2 352.641} C_DIS
LIN {X -18.7115,Y 119.2269,Z 133,A 95.0729,B 24.9391,C -1.8027,E1 24.9742,E2 350.9776} C_DIS
LIN {X -23.1954,Y 118.4371,Z 133,A 97.2584,B 24.9391,C -1.8021,E1 24.9682,E2 348.7914} C_DIS
LIN {X -26.8512,Y 117.6613,Z 133,A 98.8862,B 24.9397,C -1.7939,E1 24.9638,E2 347.181} C_DIS
LIN {X -29.9252,Y 116.9169,Z 133,A 100.4456,B 24.9397,C -1.795,E1 24.9596,E2 345.6166} C_DIS
LIN {X -32.5891,Y 116.2026,Z 133,A 101.9203,B 24.9392,C -1.8011,E1 24.9556,E2 344.1252} C_DIS
LIN {X -36.543,Y 115.0209,Z 133,A 103.802,B 24.9396,C -1.7954,E1 24.9506,E2 342.254} C_DIS
LIN {X -39.8573,Y 113.9152,Z 133,A 105.4402,B 24.9398,C -1.7924,E1 24.9463,E2 340.6197} C_DIS
LIN {X -43.7032,Y 112.4951,Z 133,A 107.3563,B 24.9401,C -1.7884,E1 24.9413,E2 338.709} C_DIS
LIN {X -46.82,Y 111.2339,Z 133,A 108.9791,B 24.9401,C -1.7873,E1 24.9371,E2 337.0851} C_DIS
LIN {X -49.4916,Y 110.0711,Z 133,A 110.3626,B 24.9403,C -1.7853,E1 24.9336,E2 335.7033} C_DIS
LIN {X -52.0301,Y 108.8942,Z 133,A 111.7999,B 24.9401,C -1.788,E1 24.9299,E2 334.2558} C_DIS
LIN {X -55.514,Y 107.1629,Z 133,A 113.7408,B 24.9401,C -1.7891,E1 24.9251,E2 332.3071} C_DIS
LIN {X -59.3796,Y 105.0698,Z 133,A 115.7731,B 24.9404,C -1.783,E1 24.9201,E2 330.2834} C_DIS
LIN {X -66.6503,Y 100.6144,Z 133,A 119.841,B 24.9409,C -1.7761,E1 24.9105,E2 326.2191} C_DIS
LIN {X -70.3351,Y 98.074,Z 133,A 121.9576,B 24.9412,C -1.7714,E1 24.9057,E2 324.1065} C_DIS
LIN {X -73.8178,Y 95.4796,Z 133,A 124.0066,B 24.9415,C -1.7664,E1 24.9011,E2 322.0618} C_DIS
LIN {X -77.0666,Y 92.8772,Z 133,A 126.009,B 24.9417,C -1.7632,E1 24.8968,E2 320.0597} C_DIS
LIN {X -80.3689,Y 90.0353,Z 133,A 128.1238,B 24.9419,C -1.7604,E1 24.8923,E2 317.9431} C_DIS
LIN {X -83.3946,Y 87.2394,Z 133,A 130.0266,B 24.9424,C -1.7534,E1 24.8885,E2 316.049} C_DIS
LIN {X -86.4339,Y 84.231,Z 133,A 132.1312,B 24.9424,C -1.7517,E1 24.8843,E2 313.9397} C_DIS
LIN {X -89.6147,Y 80.8385,Z 133,A 134.3704,B 24.9428,C -1.7474,E1 24.8801,E2 311.7007} C_DIS
LIN {X -92.3176,Y 77.7359,Z 133,A 136.2545,B 24.9433,C -1.7393,E1 24.8767,E2 309.8273} C_DIS
LIN {X -95.0063,Y 74.4266,Z 133,A 138.3079,B 24.9436,C -1.7351,E1 24.8731,E2 307.7743} C_DIS
LIN {X -97.5132,Y 71.1101,Z 133,A 140.2771,B 24.9439,C -1.7295,E1 24.8699,E2 305.809} C_DIS
LIN {X -99.8025,Y 67.8601,Z 133,A 142.6006,B 24.9431,C -1.7432,E1 24.8661,E2 303.4415} C_DIS
LIN {X -101.9688,Y 64.5587,Z 133,A 143.9984,B 24.9447,C -1.7171,E1 24.8641,E2 302.0987} C_DIS
LIN {X -103.9135,Y 61.3801,Z 133,A 145.8972,B 24.9447,C -1.7176,E1 24.8614,E2 300.189} C_DIS
LIN {X -106.0048,Y 57.6934,Z 133,A 148.6063,B 24.9431,C -1.7419,E1 24.8577,E2 297.4077} C_DIS
LIN {X -108.4722,Y 52.9065,Z 133,A 150.2762,B 24.9461,C -1.6957,E1 24.8557,E2 295.8388} C_DIS
LIN {X -109.62,Y 50.4822,Z 133,A 151.6247,B 24.9461,C -1.6951,E1 24.8541,E2 294.4845} C_DIS
LIN {X -111.0969,Y 47.1479,Z 133,A 153.5054,B 24.9461,C -1.6961,E1 24.852,E2 292.5908} C_DIS
LIN {X -112.7907,Y 42.9382,Z 133,A 155.4965,B 24.947,C -1.6824,E1 24.85,E2 290.6214} C_DIS
LIN {X -115.4278,Y 35.2359,Z 133,A 159.4532,B 24.9475,C -1.674,E1 24.8465,E2 286.662} C_DIS
LIN {X -116.4412,Y 31.7344,Z 133,A 161.337,B 24.9475,C -1.675,E1 24.845,E2 284.7649} C_DIS
LIN {X -117.3915,Y 28.0077,Z 133,A 163.0321,B 24.9481,C -1.6636,E1 24.8439,E2 283.0872} C_DIS
LIN {X -118.1391,Y 24.6694,Z 133,A 164.6676,B 24.9484,C -1.6588,E1 24.843,E2 281.4536} C_DIS
LIN {X -118.75,Y 21.5327,Z 133,A 166.2182,B 24.9487,C -1.6553,E1 24.8422,E2 279.9021} C_DIS
LIN {X -119.2846,Y 18.3395,Z 133,A 167.7242,B 24.9491,C -1.6489,E1 24.8415,E2 278.4023} C_DIS
LIN {X -119.7829,Y 14.7412,Z 133,A 169.4821,B 24.9493,C -1.6447,E1 24.8409,E2 276.6439} C_DIS
LIN {X -120.1471,Y 11.3977,Z 133,A 171.0829,B 24.9496,C -1.6397,E1 24.8404,E2 275.0456} C_DIS
LIN {X -120.3893,Y 8.461,Z 133,A 172.4559,B 24.95,C -1.634,E1 24.8401,E2 273.6779} C_DIS
LIN {X -120.5984,Y 4.5961,Z 133,A 174.4612,B 24.9499,C -1.6351,E1 24.8399,E2 271.6577} C_DIS
LIN {X -120.6805,Y 1.3412,Z 133,A 175.9523,B 24.9504,C -1.6277,E1 24.8398,E2 270.1754} C_DIS
LIN {X -120.6614,Y -2.4674,Z 133,A 177.6726,B 24.9509,C -1.618,E1 24.8398,E2 268.4677} C_DIS
LIN {X -120.5434,Y -5.878,Z 133,A 179.417,B 24.9509,C -1.618,E1 24.84,E2 266.7127} C_DIS
LIN {X -120.3293,Y -9.2795,Z 133,A -178.9876,B 24.9513,C -1.6119,E1 24.8404,E2 265.1225} C_DIS
LIN {X -119.9483,Y -13.3285,Z 133,A -177.1357,B 24.9519,C -1.6022,E1 24.8409,E2 263.2825} C_DIS
LIN {X -119.6093,Y -16.0898,Z 133,A -175.6703,B 24.9518,C -1.6042,E1 24.8414,E2 261.8036} C_DIS
LIN {X -119.0132,Y -20.0222,Z 133,A -173.8155,B 24.9522,C -1.5967,E1 24.8422,E2 259.9556} C_DIS
LIN {X -118.3251,Y -23.7552,Z 133,A -171.9729,B 24.9525,C -1.5928,E1 24.8432,E2 258.1116} C_DIS
LIN {X -117.4904,Y -27.598,Z 133,A -170.1647,B 24.953,C -1.5843,E1 24.8443,E2 256.313} C_DIS
LIN {X -116.8849,Y -30.0513,Z 133,A -169.0309,B 24.9534,C -1.5778,E1 24.8451,E2 255.1881} C_DIS
LIN {X -116.1429,Y -32.802,Z 133,A -167.638,B 24.9535,C -1.5753,E1 24.8461,E2 253.7929} C_DIS
LIN {X -115.2841,Y -35.7058,Z 133,A -165.8106,B 24.9528,C -1.5878,E1 24.8476,E2 251.9253} C_DIS
LIN {X -113.5764,Y -40.8113,Z 133,A -163.5126,B 24.9539,C -1.5689,E1 24.8497,E2 249.6593} C_DIS
LIN {X -112.3295,Y -44.1295,Z 133,A -161.725,B 24.9539,C -1.5684,E1 24.8515,E2 247.8629} C_DIS
LIN {X -110.8019,Y -47.8334,Z 133,A -159.9093,B 24.9545,C -1.5591,E1 24.8535,E2 246.0592} C_DIS
LIN {X -109.2762,Y -51.2266,Z 133,A -158.271,B 24.9551,C -1.5484,E1 24.8554,E2 244.4374} C_DIS
LIN {X -107.4411,Y -54.9686,Z 133,A -156.2119,B 24.9552,C -1.5463,E1 24.8579,E2 242.3723} C_DIS
LIN {X -105.5564,Y -58.5082,Z 133,A -154.3344,B 24.9556,C -1.5399,E1 24.8604,E2 240.5002} C_DIS
LIN {X -103.7918,Y -61.5857,Z 133,A -152.5198,B 24.9556,C -1.541,E1 24.863,E2 238.6735} C_DIS
LIN {X -102.0986,Y -64.3537,Z 133,A -150.9281,B 24.9556,C -1.5391,E1 24.8653,E2 237.078} C_DIS
LIN {X -99.7272,Y -67.9716,Z 133,A -148.8289,B 24.9558,C -1.5358,E1 24.8686,E2 234.9763} C_DIS
LIN {X -97.362,Y -71.3165,Z 133,A -146.9298,B 24.9562,C -1.5289,E1 24.8717,E2 233.0844} C_DIS
LIN {X -95.148,Y -74.2462,Z 133,A -144.947,B 24.9558,C -1.5352,E1 24.8751,E2 231.0773} C_DIS
LIN {X -91.7135,Y -78.4496,Z 133,A -142.5423,B 24.9566,C -1.5214,E1 24.8794,E2 228.6943} C_DIS
LIN {X -89.0268,Y -81.484,Z 133,A -140.4552,B 24.9565,C -1.5243,E1 24.8833,E2 226.5911} C_DIS
LIN {X -86.3803,Y -84.2855,Z 133,A -137.7663,B 24.9545,C -1.5588,E1 24.8888,E2 223.8084} C_DIS
LIN {X -81.476,Y -89.0342,Z 133,A -135.6593,B 24.9578,C -1.5011,E1 24.8928,E2 221.8301} C_DIS
LIN {X -78.6124,Y -91.5732,Z 133,A -133.6692,B 24.9576,C -1.5052,E1 24.897,E2 219.8225} C_DIS
LIN {X -74.8537,Y -94.6706,Z 133,A -131.6793,B 24.9586,C -1.4865,E1 24.9013,E2 217.8696} C_DIS
LIN {X -72.3076,Y -96.6297,Z 133,A -129.8579,B 24.958,C -1.497,E1 24.9054,E2 216.0168} C_DIS
LIN {X -69.007,Y -99.0123,Z 133,A -128.0925,B 24.9586,C -1.4862,E1 24.9094,E2 214.2709} C_DIS
LIN {X -66.1616,Y -100.9369,Z 133,A -126.3478,B 24.9585,C -1.4886,E1 24.9134,E2 212.5147} C_DIS
LIN {X -63.0467,Y -102.9101,Z 133,A -124.6026,B 24.9586,C -1.4857,E1 24.9176,E2 210.7709} C_DIS
LIN {X -59.5923,Y -104.9491,Z 133,A -122.5695,B 24.9585,C -1.4888,E1 24.9225,E2 208.7244} C_DIS
LIN {X -55.5704,Y -107.1333,Z 133,A -120.2824,B 24.9583,C -1.4911,E1 24.9282,E2 206.4255} C_DIS
LIN {X -51.5099,Y -109.1431,Z 133,A -118.1969,B 24.9587,C -1.4855,E1 24.9334,E2 204.3479} C_DIS
LIN {X -48.0187,Y -110.7218,Z 133,A -116.5708,B 24.9593,C -1.4747,E1 24.9375,E2 202.7436} C_DIS
LIN {X -44.3565,Y -112.2414,Z 133,A -114.7111,B 24.9594,C -1.4717,E1 24.9423,E2 200.8869} C_DIS
LIN {X -40.7469,Y -113.5996,Z 133,A -112.8332,B 24.9594,C -1.4722,E1 24.9473,E2 199.0039} C_DIS
LIN {X -37.3029,Y -114.7778,Z 133,A -111.2074,B 24.9597,C -1.4661,E1 24.9515,E2 197.3897} C_DIS
LIN {X -34.9875,Y -115.5037,Z 133,A -109.8716,B 24.9593,C -1.4737,E1 24.9552,E2 196.0334} C_DIS
LIN {X -31.4911,Y -116.506,Z 133,A -108.1872,B 24.9595,C -1.4706,E1 24.9597,E2 194.3538} C_DIS
LIN {X -27.9444,Y -117.4068,Z 133,A -106.4364,B 24.9595,C -1.4702,E1 24.9644,E2 192.6013} C_DIS
LIN {X -24.5411,Y -118.1652,Z 133,A -104.9626,B 24.96,C -1.4611,E1 24.9684,E2 191.1475} C_DIS
LIN {X -21.6969,Y -118.7207,Z 133,A -103.3531,B 24.9594,C -1.4714,E1 24.9729,E2 189.5118} C_DIS
LIN {X -17.8307,Y -119.3635,Z 133,A -101.367,B 24.9591,C -1.4767,E1 24.9784,E2 187.5113} C_DIS
LIN {X -12.3153,Y -120.0581,Z 133,A -98.9954,B 24.9599,C -1.4638,E1 24.9849,E2 185.1687} C_DIS
LIN {X -8.8849,Y -120.3582,Z 133,A -97.0131,B 24.959,C -1.4801,E1 24.9905,E2 183.147} C_DIS
LIN {X -0.2657,Y -120.6871,Z 133,A -93.2452,B 24.9598,C -1.4652,E1 25.001,E2 179.414} C_DIS
LIN {X -0.2657,Y -120.6871,Z 133,A -93.2452,B 24.9598,C -1.4652,E1 25.001,E2 179.414} C_DIS
Enddeposition()
LIN {X 0.8527,Y -119.8469,Z 133,A -92.588,B 24.9586,C -1.4857,E1 25.0029,E2 178.7081} C_DIS
Startdeposition()
$VEL.CP = VEL_PRINT
LIN {X -2.5012,Y -119.8238,Z 133,A -95.0926,B 24.961,C -1.4435,E1 24.9957,E2 181.3126} C_DIS
LIN {X -5.9122,Y -119.7038,Z 133,A -96.6231,B 24.9607,C -1.448,E1 24.9914,E2 182.8328} C_DIS
LIN {X -9.329,Y -119.4866,Z 133,A -98.2427,B 24.9607,C -1.4488,E1 24.9869,E2 184.4512} C_DIS
LIN {X -13.2401,Y -119.1162,Z 133,A -100.115,B 24.9607,C -1.4493,E1 24.9817,E2 186.3234} C_DIS
LIN {X -16.645,Y -118.6883,Z 133,A -101.7713,B 24.9607,C -1.4489,E1 24.9771,E2 187.982} C_DIS
LIN {X -19.0521,Y -118.3267,Z 133,A -102.9434,B 24.9607,C -1.4488,E1 24.9739,E2 189.1553} C_DIS
LIN {X -21.9423,Y -117.8256,Z 133,A -104.5026,B 24.961,C -1.4422,E1 24.9695,E2 190.7318} C_DIS
LIN {X -25.7913,Y -117.042,Z 133,A -106.321,B 24.9608,C -1.4457,E1 24.9646,E2 192.5439} C_DIS
LIN {X -29.1271,Y -116.2558,Z 133,A -107.831,B 24.9605,C -1.4524,E1 24.9605,E2 194.0401} C_DIS
LIN {X -31.9687,Y -115.5075,Z 133,A -109.3938,B 24.9608,C -1.4462,E1 24.9563,E2 195.6201} C_DIS
LIN {X -35.2637,Y -114.5442,Z 133,A -110.9686,B 24.9606,C -1.4504,E1 24.9521,E2 197.1877} C_DIS
LIN {X -39.1054,Y -113.2899,Z 133,A -112.8422,B 24.9604,C -1.4546,E1 24.9471,E2 199.0548} C_DIS
LIN {X -41.9742,Y -112.258,Z 133,A -114.3381,B 24.9604,C -1.4542,E1 24.9432,E2 200.5547} C_DIS
LIN {X -45.4262,Y -110.9078,Z 133,A -116.1949,B 24.9604,C -1.4521,E1 24.9384,E2 202.4203} C_DIS
LIN {X -48.5735,Y -109.5652,Z 133,A -117.8454,B 24.9604,C -1.4533,E1 24.9341,E2 204.072} C_DIS
LIN {X -51.6878,Y -108.1303,Z 133,A -119.3741,B 24.9601,C -1.4602,E1 24.9303,E2 205.5883} C_DIS
LIN {X -55.196,Y -106.3846,Z 133,A -121.392,B 24.9603,C -1.4561,E1 24.9252,E2 207.6212} C_DIS
LIN {X -59.1503,Y -104.2379,Z 133,A -123.5059,B 24.96,C -1.4607,E1 24.9201,E2 209.7302} C_DIS
LIN {X -62.2409,Y -102.4217,Z 133,A -125.0566,B 24.9595,C -1.4705,E1 24.9164,E2 211.2624} C_DIS
LIN {X -64.544,Y -100.9859,Z 133,A -126.5027,B 24.9597,C -1.4659,E1 24.913,E2 212.7239} C_DIS
LIN {X -67.8002,Y -98.8297,Z 133,A -128.3916,B 24.9597,C -1.468,E1 24.9086,E2 214.6142} C_DIS
LIN {X -71.0004,Y -96.5558,Z 133,A -130.264,B 24.9594,C -1.4715,E1 24.9043,E2 216.4849} C_DIS
LIN {X -74.3297,Y -94.018,Z 133,A -132.3384,B 24.9594,C -1.4719,E1 24.8997,E2 218.5659} C_DIS
LIN {X -77.7278,Y -91.2284,Z 133,A -134.4624,B 24.9592,C -1.475,E1 24.8952,E2 220.6906} C_DIS
LIN {X -80.8997,Y -88.4272,Z 133,A -136.3547,B 24.9587,C -1.4848,E1 24.8913,E2 222.5672} C_DIS
LIN {X -83.7216,Y -85.7612,Z 133,A -138.3484,B 24.9588,C -1.4827,E1 24.8873,E2 224.5742} C_DIS
LIN {X -86.798,Y -82.6453,Z 133,A -140.4025,B 24.9585,C -1.489,E1 24.8833,E2 226.6221} C_DIS
LIN {X -89.4649,Y -79.7514,Z 133,A -142.3414,B 24.9584,C -1.4908,E1 24.8796,E2 228.5653} C_DIS
LIN {X -92.3364,Y -76.4078,Z 133,A -144.413,B 24.958,C -1.4973,E1 24.8759,E2 230.6309} C_DIS
LIN {X -94.784,Y -73.3494,Z 133,A -146.2391,B 24.9576,C -1.5038,E1 24.8728,E2 232.4501} C_DIS
LIN {X -97.1343,Y -70.2081,Z 133,A -148.2088,B 24.9576,C -1.5045,E1 24.8695,E2 234.4278} C_DIS
LIN {X -99.3846,Y -66.9839,Z 133,A -150.051,B 24.9572,C -1.5109,E1 24.8666,E2 236.2637} C_DIS
LIN {X -101.2588,Y -64.1157,Z 133,A -151.6016,B 24.9568,C -1.519,E1 24.8643,E2 237.803} C_DIS
LIN {X -102.8405,Y -61.5472,Z 133,A -153.1547,B 24.9568,C -1.5181,E1 24.862,E2 239.3662} C_DIS
LIN {X -104.7511,Y -58.2351,Z 133,A -154.9988,B 24.9566,C -1.5224,E1 24.8595,E2 241.2095} C_DIS
LIN {X -106.3848,Y -55.1958,Z 133,A -156.7484,B 24.9566,C -1.5228,E1 24.8572,E2 242.9677} C_DIS
LIN {X -108.131,Y -51.6864,Z 133,A -158.5446,B 24.9561,C -1.5314,E1 24.855,E2 244.753} C_DIS
LIN {X -109.7713,Y -48.1082,Z 133,A -160.5004,B 24.9559,C -1.5337,E1 24.8527,E2 246.7141} C_DIS
LIN {X -111.2802,Y -44.5044,Z 133,A -162.2184,B 24.9552,C -1.5456,E1 24.8509,E2 248.4134} C_DIS
LIN {X -112.3367,Y -41.7638,Z 133,A -163.6588,B 24.9551,C -1.5482,E1 24.8495,E2 249.8555} C_DIS
LIN {X -113.4848,Y -38.5403,Z 133,A -165.2639,B 24.9547,C -1.5544,E1 24.848,E2 251.4549} C_DIS
LIN {X -114.5778,Y -35.1538,Z 133,A -167.0745,B 24.9547,C -1.555,E1 24.8465,E2 253.2746} C_DIS
LIN {X -115.6424,Y -31.4823,Z 133,A -168.8518,B 24.9542,C -1.5628,E1 24.8452,E2 255.0438} C_DIS
LIN {X -116.3851,Y -28.6092,Z 133,A -170.2035,B 24.9538,C -1.57,E1 24.8443,E2 256.386} C_DIS
LIN {X -117.207,Y -25.0266,Z 133,A -172.1592,B 24.954,C -1.5672,E1 24.8431,E2 258.3599} C_DIS
LIN {X -117.9161,Y -21.442,Z 133,A -173.8762,B 24.9536,C -1.574,E1 24.8422,E2 260.0709} C_DIS
LIN {X -118.4788,Y -18.0749,Z 133,A -175.511,B 24.9533,C -1.5791,E1 24.8415,E2 261.7033} C_DIS
LIN {X -119.0075,Y -14.1765,Z 133,A -177.3006,B 24.9527,C -1.589,E1 24.8408,E2 263.48} C_DIS
LIN {X -119.3667,Y -10.7641,Z 133,A -179.1349,B 24.9529,C -1.5861,E1 24.8403,E2 265.332} C_DIS
LIN {X -119.6279,Y -7.2818,Z 133,A 179.3009,B 24.9523,C -1.596,E1 24.84,E2 266.8822} C_DIS
LIN {X -119.8134,Y -2.9455,Z 133,A 177.1453,B 24.9521,C -1.5994,E1 24.8398,E2 269.0427} C_DIS
LIN {X -119.8472,Y 0.8693,Z 133,A 175.2696,B 24.9518,C -1.6032,E1 24.8398,E2 270.9206} C_DIS
LIN {X -119.7297,Y 5.3913,Z 133,A 173.0921,B 24.9515,C -1.6096,E1 24.84,E2 273.0959} C_DIS
LIN {X -119.4883,Y 9.306,Z 133,A 171.3877,B 24.9506,C -1.6229,E1 24.8403,E2 274.7789} C_DIS
LIN {X -119.1717,Y 12.7269,Z 133,A 169.607,B 24.9506,C -1.6225,E1 24.8408,E2 276.5712} C_DIS
LIN {X -118.6912,Y 16.6246,Z 133,A 167.8042,B 24.9501,C -1.6318,E1 24.8415,E2 278.3627} C_DIS
LIN {X -118.3289,Y 19.039,Z 133,A 166.6207,B 24.9499,C -1.6349,E1 24.842,E2 279.5458} C_DIS
LIN {X -117.8274,Y 21.9327,Z 133,A 165.0487,B 24.9501,C -1.6324,E1 24.8428,E2 281.133} C_DIS
LIN {X -117.0457,Y 25.774,Z 133,A 163.1955,B 24.9496,C -1.6394,E1 24.8439,E2 282.9806} C_DIS
LIN {X -116.1394,Y 29.5863,Z 133,A 161.4042,B 24.9491,C -1.6489,E1 24.845,E2 284.7597} C_DIS
LIN {X -114.9678,Y 33.8544,Z 133,A 159.3216,B 24.9485,C -1.657,E1 24.8466,E2 286.8349} C_DIS
LIN {X -113.9277,Y 37.211,Z 133,A 157.4956,B 24.9485,C -1.6562,E1 24.8482,E2 288.6734} C_DIS
LIN {X -112.8388,Y 40.3899,Z 133,A 155.8825,B 24.9483,C -1.661,E1 24.8497,E2 290.2842} C_DIS
LIN {X -111.6342,Y 43.6082,Z 133,A 154.2735,B 24.9479,C -1.6676,E1 24.8513,E2 291.8866} C_DIS
LIN {X -110.1534,Y 47.2246,Z 133,A 152.4722,B 24.9474,C -1.6762,E1 24.8532,E2 293.6774} C_DIS
LIN {X -108.7545,Y 50.3603,Z 133,A 150.7801,B 24.9472,C -1.6791,E1 24.8551,E2 295.3718} C_DIS
LIN {X -107.4676,Y 53.0509,Z 133,A 149.397,B 24.9468,C -1.6852,E1 24.8568,E2 296.7479} C_DIS
LIN {X -105.4519,Y 56.9586,Z 133,A 147.0845,B 24.9469,C -1.6826,E1 24.8598,E2 299.0789} C_DIS
LIN {X -103.2958,Y 60.7791,Z 133,A 145.1587,B 24.9461,C -1.696,E1 24.8625,E2 300.9828} C_DIS
LIN {X -101.7809,Y 63.2837,Z 133,A 143.738,B 24.9459,C -1.6991,E1 24.8646,E2 302.4033} C_DIS
LIN {X -99.9445,Y 66.1461,Z 133,A 141.9986,B 24.9459,C -1.699,E1 24.8672,E2 304.1518} C_DIS
LIN {X -97.7021,Y 69.4158,Z 133,A 140.0595,B 24.9457,C -1.7024,E1 24.8703,E2 306.0923} C_DIS
LIN {X -95.3763,Y 72.578,Z 133,A 138.1713,B 24.9454,C -1.7071,E1 24.8735,E2 307.9784} C_DIS
LIN {X -92.6446,Y 76.0347,Z 133,A 136.036,B 24.9451,C -1.7115,E1 24.8772,E2 310.1132} C_DIS
LIN {X -89.7864,Y 79.3884,Z 133,A 133.9813,B 24.9446,C -1.7192,E1 24.881,E2 312.1589} C_DIS
LIN {X -87.1072,Y 82.3195,Z 133,A 132.0258,B 24.9445,C -1.7215,E1 24.8847,E2 314.1173} C_DIS
LIN {X -84.225,Y 85.2666,Z 133,A 130.0252,B 24.9442,C -1.7251,E1 24.8886,E2 316.1179} C_DIS
LIN {X -81.2159,Y 88.1368,Z 133,A 128.0912,B 24.9438,C -1.7321,E1 24.8925,E2 318.0431} C_DIS
LIN {X -77.9024,Y 91.0802,Z 133,A 125.936,B 24.9436,C -1.7354,E1 24.8971,E2 320.1989} C_DIS
LIN {X -74.8898,Y 93.5717,Z 133,A 124.0812,B 24.9432,C -1.7402,E1 24.9011,E2 322.0493} C_DIS
LIN {X -72.1806,Y 95.6773,Z 133,A 122.3882,B 24.9432,C -1.7415,E1 24.9049,E2 323.7455} C_DIS
LIN {X -68.7722,Y 98.1558,Z 133,A 120.5798,B 24.9423,C -1.7545,E1 24.9089,E2 325.5292} C_DIS
LIN {X -66.5823,Y 99.6538,Z 133,A 119.1565,B 24.9426,C -1.7504,E1 24.9122,E2 326.9671} C_DIS
LIN {X -63.1313,Y 101.8755,Z 133,A 117.1961,B 24.9423,C -1.7542,E1 24.9168,E2 328.9246} C_DIS
LIN {X -59.8977,Y 103.8096,Z 133,A 115.3536,B 24.9423,C -1.7557,E1 24.9213,E2 330.7691} C_DIS
LIN {X -56.482,Y 105.707,Z 133,A 113.6084,B 24.9417,C -1.7642,E1 24.9255,E2 332.4989} C_DIS
LIN {X -53.8775,Y 107.0568,Z 133,A 112.1898,B 24.9416,C -1.7659,E1 24.9291,E2 333.9174} C_DIS
LIN {X -51.2382,Y 108.3454,Z 133,A 110.6094,B 24.9419,C -1.7605,E1 24.9331,E2 335.5148} C_DIS
LIN {X -48.1157,Y 109.7681,Z 133,A 109.1158,B 24.9413,C -1.7693,E1 24.9368,E2 336.9909} C_DIS
LIN {X -45.4132,Y 110.913,Z 133,A 107.5963,B 24.9415,C -1.7663,E1 24.9408,E2 338.5211} C_DIS
LIN {X -41.7547,Y 112.3401,Z 133,A 105.796,B 24.9411,C -1.7722,E1 24.9455,E2 340.3111} C_DIS
LIN {X -38.0015,Y 113.6644,Z 133,A 104.0885,B 24.9404,C -1.7831,E1 24.9499,E2 341.9959} C_DIS
LIN {X -34.7817,Y 114.6915,Z 133,A 102.2951,B 24.9408,C -1.7772,E1 24.9547,E2 343.8067} C_DIS
LIN {X -31.4806,Y 115.6428,Z 133,A 100.638,B 24.9408,C -1.7783,E1 24.9592,E2 345.4638} C_DIS
LIN {X -28.6391,Y 116.3778,Z 133,A 99.2299,B 24.9407,C -1.7795,E1 24.963,E2 346.871} C_DIS
LIN {X -25.7659,Y 117.0475,Z 133,A 97.7148,B 24.9409,C -1.7761,E1 24.9671,E2 348.396} C_DIS
LIN {X -21.9187,Y 117.8301,Z 133,A 95.7937,B 24.9409,C -1.7757,E1 24.9724,E2 350.3203} C_DIS
LIN {X -19.0304,Y 118.3302,Z 133,A 94.5946,B 24.9402,C -1.7857,E1 24.9757,E2 351.4968} C_DIS
LIN {X -15.6375,Y 118.8245,Z 133,A 92.8224,B 24.9406,C -1.7808,E1 24.9806,E2 353.2819} C_DIS
LIN {X -11.6924,Y 119.2782,Z 133,A 90.9947,B 24.9403,C -1.785,E1 24.9856,E2 355.1008} C_DIS
LIN {X -8.2886,Y 119.5628,Z 133,A 89.3005,B 24.9404,C -1.783,E1 24.9904,E2 356.8005} C_DIS
LIN {X -5.2731,Y 119.7349,Z 133,A 87.7181,B 24.9408,C -1.7773,E1 24.9948,E2 358.3968} C_DIS
LIN {X -1.4508,Y 119.8418,Z 133,A 85.9885,B 24.9405,C -1.7822,E1 24.9996,E2 360.1149} C_DIS
LIN {X 2.4735,Y 119.8243,Z 133,A 84.1136,B 24.9405,C -1.7825,E1 25.0049,E2 361.9888} C_DIS
LIN {X 5.8898,Y 119.7049,Z 133,A 82.5822,B 24.9401,C -1.7873,E1 25.0091,E2 363.5085} C_DIS
LIN {X 9.3099,Y 119.488,Z 133,A 80.9896,B 24.94,C -1.7893,E1 25.0135,E2 365.0957} C_DIS
LIN {X 12.7393,Y 119.1704,Z 133,A 79.2219,B 24.9404,C -1.7836,E1 25.0185,E2 366.8757} C_DIS
LIN {X 16.6318,Y 118.6902,Z 133,A 77.433,B 24.9401,C -1.7871,E1 25.0234,E2 368.655} C_DIS
LIN {X 19.0427,Y 118.3282,Z 133,A 76.2615,B 24.9401,C -1.7864,E1 25.0266,E2 369.8269} C_DIS
LIN {X 21.9536,Y 117.8234,Z 133,A 74.6952,B 24.9407,C -1.7788,E1 25.031,E2 371.4094} C_DIS
LIN {X 25.7851,Y 117.0433,Z 133,A 72.8885,B 24.9406,C -1.7808,E1 25.0359,E2 373.2091} C_DIS
LIN {X 29.1236,Y 116.2567,Z 133,A 71.3803,B 24.9402,C -1.7859,E1 25.0399,E2 374.703} C_DIS
LIN {X 31.9651,Y 115.5085,Z 133,A 69.8213,B 24.9408,C -1.7779,E1 25.0442,E2 376.2786} C_DIS
LIN {X 35.2591,Y 114.5456,Z 133,A 68.2498,B 24.9406,C -1.7798,E1 25.0484,E2 377.8427} C_DIS
LIN {X 38.9944,Y 113.3284,Z 133,A 66.444,B 24.9406,C -1.7816,E1 25.0531,E2 379.6409} C_DIS
LIN {X 42.4908,Y 112.0646,Z 133,A 64.5166,B 24.9411,C -1.7729,E1 25.0582,E2 381.5847} C_DIS
LIN {X 45.8698,Y 110.7238,Z 133,A 62.9263,B 24.9408,C -1.778,E1 25.0623,E2 383.1594} C_DIS
LIN {X 48.5668,Y 109.5682,Z 133,A 61.4048,B 24.9412,C -1.7708,E1 25.0662,E2 384.6941} C_DIS
LIN {X 51.6922,Y 108.1282,Z 133,A 59.8782,B 24.941,C -1.7744,E1 25.0701,E2 386.2084} C_DIS
LIN {X 54.9096,Y 106.5324,Z 133,A 57.9836,B 24.9417,C -1.7638,E1 25.0748,E2 388.1228} C_DIS
LIN {X 59.0939,Y 104.2701,Z 133,A 55.7861,B 24.9417,C -1.7642,E1 25.0802,E2 390.313} C_DIS
LIN {X 62.0485,Y 102.5382,Z 133,A 54.2415,B 24.9415,C -1.7661,E1 25.0839,E2 391.8484} C_DIS
LIN {X 65.353,Y 100.4652,Z 133,A 52.2997,B 24.942,C -1.7595,E1 25.0885,E2 393.7995} C_DIS
LIN {X 68.2179,Y 98.5423,Z 133,A 50.7787,B 24.9418,C -1.7628,E1 25.0919,E2 395.3076} C_DIS
LIN {X 71.1145,Y 96.4719,Z 133,A 48.9653,B 24.9423,C -1.7545,E1 25.0961,E2 397.134} C_DIS
LIN {X 74.3979,Y 93.9641,Z 133,A 46.9815,B 24.9426,C -1.7505,E1 25.1004,E2 399.1201} C_DIS
LIN {X 77.7256,Y 91.2302,Z 133,A 44.8984,B 24.9429,C -1.7453,E1 25.1049,E2 401.2074} C_DIS
LIN {X 80.843,Y 88.4792,Z 133,A 43.0534,B 24.9427,C -1.748,E1 25.1087,E2 403.0386} C_DIS
LIN {X 83.7463,Y 85.737,Z 133,A 41.038,B 24.9433,C -1.7389,E1 25.1128,E2 405.0671} C_DIS
LIN {X 86.8069,Y 82.6359,Z 133,A 39.0079,B 24.9435,C -1.7369,E1 25.1168,E2 407.0934} C_DIS
LIN {X 89.4626,Y 79.7539,Z 133,A 37.092,B 24.9439,C -1.7305,E1 25.1204,E2 409.0157} C_DIS
LIN {X 92.3325,Y 76.4126,Z 133,A 35.0424,B 24.944,C -1.7282,E1 25.124,E2 411.0614} C_DIS
LIN {X 94.7837,Y 73.3497,Z 133,A 33.2024,B 24.9442,C -1.7253,E1 25.1272,E2 412.8996} C_DIS
LIN {X 97.172,Y 70.1563,Z 133,A 31.3652,B 24.9443,C -1.7239,E1 25.1303,E2 414.7315} C_DIS
LIN {X 98.8423,Y 67.782,Z 133,A 29.9097,B 24.9447,C -1.717,E1 25.1326,E2 416.1959} C_DIS
LIN {X 100.991,Y 64.5359,Z 133,A 28.0701,B 24.945,C -1.7132,E1 25.1354,E2 418.0354} C_DIS
LIN {X 102.8031,Y 61.61,Z 133,A 26.4066,B 24.9453,C -1.7079,E1 25.1378,E2 419.703} C_DIS
LIN {X 104.7577,Y 58.2231,Z 133,A 24.5685,B 24.9456,C -1.7042,E1 25.1403,E2 421.54} C_DIS
LIN {X 106.5496,Y 54.8758,Z 133,A 22.8939,B 24.9455,C -1.706,E1 25.1425,E2 423.2018} C_DIS
LIN {X 107.7238,Y 52.5321,Z 133,A 21.6293,B 24.9457,C -1.7018,E1 25.1441,E2 424.4693} C_DIS
LIN {X 109.1765,Y 49.442,Z 133,A 19.908,B 24.9463,C -1.6928,E1 25.1461,E2 426.2026} C_DIS
LIN {X 110.3472,Y 46.7715,Z 133,A 18.5774,B 24.9463,C -1.6918,E1 25.1476,E2 427.5283} C_DIS
LIN {X 111.6406,Y 43.5916,Z 133,A 16.8607,B 24.9469,C -1.6833,E1 25.1494,E2 429.2556} C_DIS
LIN {X 113.0109,Y 39.9114,Z 133,A 14.9159,B 24.9475,C -1.6743,E1 25.1512,E2 431.2106} C_DIS
LIN {X 114.1878,Y 36.4004,Z 133,A 13.3134,B 24.9473,C -1.6771,E1 25.1526,E2 432.7975} C_DIS
LIN {X 115.108,Y 33.3759,Z 133,A 11.7988,B 24.9476,C -1.6723,E1 25.1538,E2 434.3148} C_DIS
LIN {X 116.0178,Y 30.0663,Z 133,A 10.0976,B 24.9481,C -1.6642,E1 25.155,E2 436.0252} C_DIS
LIN {X 116.7339,Y 27.1547,Z 133,A 8.7684,B 24.9481,C -1.6648,E1 25.1559,E2 437.3454} C_DIS
LIN {X 117.4529,Y 23.8447,Z 133,A 7.1517,B 24.9484,C -1.6599,E1 25.1568,E2 438.9643} C_DIS
LIN {X 118.1692,Y 19.9954,Z 133,A 5.5303,B 24.948,C -1.6662,E1 25.1576,E2 440.5614} C_DIS
LIN {X 118.5834,Y 17.3824,Z 133,A 3.9419,B 24.9492,C -1.6462,E1 25.1583,E2 442.1875} C_DIS
LIN {X 119.0745,Y 13.6138,Z 133,A 2.1657,B 24.9495,C -1.6423,E1 25.1589,E2 443.9623} C_DIS
LIN {X 119.4092,Y 10.2599,Z 133,A 0.5803,B 24.9497,C -1.6384,E1 25.1593,E2 445.5476} C_DIS
LIN {X 119.6939,Y 6.1122,Z 133,A -1.3938,B 24.9501,C -1.6326,E1 25.1596,E2 447.5237} C_DIS
LIN {X 119.8262,Y 2.3604,Z 133,A -3.0668,B 24.9501,C -1.6326,E1 25.1598,E2 449.1865} C_DIS
LIN {X 119.8474,Y -0.832,Z 133,A -4.7243,B 24.9508,C -1.6212,E1 25.1598,E2 450.8611} C_DIS
LIN {X 119.7466,Y -4.9691,Z 133,A -6.6129,B 24.9508,C -1.6191,E1 25.1596,E2 452.7434} C_DIS
LIN {X 119.5216,Y -8.8507,Z 133,A -8.4606,B 24.9512,C -1.6136,E1 25.1593,E2 454.5932} C_DIS
LIN {X 119.17,Y -12.7427,Z 133,A -10.3579,B 24.9517,C -1.606,E1 25.1588,E2 456.4971} C_DIS
LIN {X 118.6906,Y -16.6286,Z 133,A -12.1322,B 24.9517,C -1.6047,E1 25.1581,E2 458.2641} C_DIS
LIN {X 118.3292,Y -19.0366,Z 133,A -13.3457,B 24.9521,C -1.5984,E1 25.1576,E2 459.4852} C_DIS
LIN {X 117.8248,Y -21.9464,Z 133,A -14.8525,B 24.9527,C -1.5891,E1 25.1568,E2 461.0051} C_DIS
LIN {X 117.014,Y -25.9208,Z 133,A -16.707,B 24.9528,C -1.587,E1 25.1558,E2 462.8539} C_DIS
LIN {X 116.2566,Y -29.1241,Z 133,A -18.1525,B 24.9528,C -1.5882,E1 25.1548,E2 464.2881} C_DIS
LIN {X 115.5087,Y -31.9642,Z 133,A -19.5911,B 24.9531,C -1.582,E1 25.1538,E2 465.7331} C_DIS
LIN {X 114.5466,Y -35.256,Z 133,A -21.2669,B 24.9535,C -1.5749,E1 25.1524,E2 467.416} C_DIS
LIN {X 113.3296,Y -38.9909,Z 133,A -23.0536,B 24.9536,C -1.5734,E1 25.1508,E2 469.1961} C_DIS
LIN {X 112.02,Y -42.6099,Z 133,A -25.0305,B 24.9544,C -1.5609,E1 25.1489,E2 471.1915} C_DIS
LIN {X 110.7214,Y -45.8757,Z 133,A -26.5393,B 24.9542,C -1.5641,E1 25.1473,E2 472.6844} C_DIS
LIN {X 109.5649,Y -48.5741,Z 133,A -28.0815,B 24.9548,C -1.5529,E1 25.1456,E2 474.2446} C_DIS
LIN {X 108.0674,Y -51.8192,Z 133,A -29.6394,B 24.9547,C -1.5551,E1 25.1438,E2 475.7889} C_DIS
LIN {X 106.3901,Y -55.1857,Z 133,A -31.5375,B 24.9553,C -1.5447,E1 25.1413,E2 477.7014} C_DIS
LIN {X 104.7551,Y -58.2278,Z 133,A -33.1748,B 24.9555,C -1.5405,E1 25.1391,E2 479.3401} C_DIS
LIN {X 102.7147,Y -61.7572,Z 133,A -35.1186,B 24.9559,C -1.535,E1 25.1364,E2 481.2869} C_DIS
LIN {X 100.4584,Y -65.3634,Z 133,A -37.1559,B 24.9562,C -1.5289,E1 25.1333,E2 483.3283} C_DIS
LIN {X 98.5452,Y -68.2138,Z 133,A -38.6687,B 24.9562,C -1.5305,E1 25.131,E2 484.8298} C_DIS
LIN {X 96.4641,Y -71.1251,Z 133,A -40.4308,B 24.9565,C -1.5233,E1 25.1281,E2 486.6004} C_DIS
LIN {X 94.0243,Y -74.3218,Z 133,A -42.4354,B 24.9571,C -1.514,E1 25.1246,E2 488.6174} C_DIS
LIN {X 91.2304,Y -77.7254,Z 133,A -44.5398,B 24.9574,C -1.5085,E1 25.1208,E2 490.7253} C_DIS
LIN {X 88.4618,Y -80.8619,Z 133,A -46.3942,B 24.9573,C -1.5103,E1 25.1174,E2 492.567} C_DIS
LIN {X 85.7745,Y -83.7081,Z 133,A -48.3844,B 24.9579,C -1.4998,E1 25.1135,E2 494.5734} C_DIS
LIN {X 82.6426,Y -86.8006,Z 133,A -50.4288,B 24.9579,C -1.4976,E1 25.1094,E2 496.6146} C_DIS
LIN {X 79.7426,Y -89.4727,Z 133,A -52.3477,B 24.9583,C -1.4915,E1 25.1055,E2 498.5402} C_DIS
LIN {X 76.4037,Y -92.3398,Z 133,A -54.3907,B 24.9584,C -1.4896,E1 25.1011,E2 500.5797} C_DIS
LIN {X 73.3526,Y -94.7814,Z 133,A -56.2825,B 24.9587,C -1.4844,E1 25.0969,E2 502.4768} C_DIS
LIN {X 70.2003,Y -97.14,Z 133,A -58.0435,B 24.9587,C -1.4862,E1 25.093,E2 504.2273} C_DIS
LIN {X 67.7991,Y -98.8304,Z 133,A -59.5181,B 24.959,C -1.4799,E1 25.0896,E2 505.7117} C_DIS
LIN {X 64.5385,Y -100.9894,Z 133,A -61.3716,B 24.9591,C -1.4769,E1 25.0853,E2 507.566} C_DIS
LIN {X 61.6204,Y -102.7968,Z 133,A -63.031,B 24.9594,C -1.4729,E1 25.0813,E2 509.2297} C_DIS
LIN {X 58.2216,Y -104.7585,Z 133,A -64.8802,B 24.9594,C -1.4708,E1 25.0768,E2 511.0784} C_DIS
LIN {X 55.1479,Y -106.4099,Z 133,A -66.4976,B 24.9595,C -1.4703,E1 25.0728,E2 512.6924} C_DIS
LIN {X 52.5445,Y -107.7176,Z 133,A -67.8508,B 24.9595,C -1.4699,E1 25.0694,E2 514.043} C_DIS
LIN {X 49.4434,Y -109.1759,Z 133,A -69.4439,B 24.9595,C -1.4695,E1 25.0654,E2 515.6331} C_DIS
LIN {X 46.7625,Y -110.351,Z 133,A -70.858,B 24.9597,C -1.4666,E1 25.0618,E2 517.0505} C_DIS
LIN {X 43.4689,Y -111.6883,Z 133,A -72.6396,B 24.96,C -1.4603,E1 25.0571,E2 518.8429} C_DIS
LIN {X 39.9032,Y -113.0137,Z 133,A -74.4006,B 24.96,C -1.4606,E1 25.0525,E2 520.5997} C_DIS
LIN {X 36.7071,Y -114.0897,Z 133,A -76.0198,B 24.9602,C -1.4583,E1 25.0482,E2 522.2213} C_DIS
LIN {X 33.3643,Y -115.1114,Z 133,A -77.6995,B 24.9602,C -1.4559,E1 25.0437,E2 523.9036} C_DIS
LIN {X 30.0521,Y -116.0214,Z 133,A -79.2936,B 24.9602,C -1.4564,E1 25.0394,E2 525.494} C_DIS
LIN {X 27.2048,Y -116.7226,Z 133,A -80.715,B 24.9604,C -1.4541,E1 25.0355,E2 526.9189} C_DIS
LIN {X 23.85,Y -117.4518,Z 133,A -82.3558,B 24.9604,C -1.4527,E1 25.0311,E2 528.561} C_DIS
LIN {X 19.9569,Y -118.1757,Z 133,A -83.9996,B 24.9599,C -1.4628,E1 25.0266,E2 530.179} C_DIS
LIN {X 17.5572,Y -118.5586,Z 133,A -85.5367,B 24.9609,C -1.4444,E1 25.0223,E2 531.7583} C_DIS
LIN {X 13.6978,Y -119.0645,Z 133,A -87.3236,B 24.9608,C -1.4467,E1 25.0173,E2 533.5384} C_DIS
LIN {X 10.2926,Y -119.4065,Z 133,A -88.953,B 24.9608,C -1.4461,E1 25.0128,E2 535.1681} C_DIS
LIN {X 6.4234,Y -119.6784,Z 133,A -90.8583,B 24.961,C -1.4429,E1 25.0075,E2 537.0802} C_DIS
LIN {X 2.9876,Y -119.8122,Z 133,A -92.487,B 24.961,C -1.4431,E1 25.0029,E2 538.7081} C_DIS
LIN {X 2.9876,Y -119.8122,Z 133,A -92.487,B 24.961,C -1.4431,E1 25.0029,E2 538.7081} C_DIS
Enddeposition()
LIN {X 0.8896,Y -125.3254,Z 134,A -92.9503,B 24.9643,C -1.3803,E1 25.0012,E2 539.3201} C_DIS
Startdeposition()
$VEL.CP = VEL_PRINT
LIN {X 3.4129,Y -125.2819,Z 134,A -91.4465,B 24.9634,C -1.3978,E1 25.0055,E2 537.7751} C_DIS
LIN {X 7.0305,Y -125.1328,Z 134,A -89.7858,B 24.9634,C -1.3987,E1 25.0102,E2 536.1128} C_DIS
LIN {X 10.4233,Y -124.8942,Z 134,A -88.2591,B 24.9634,C -1.3981,E1 25.0144,E2 534.5883} C_DIS
LIN {X 14.5538,Y -124.4807,Z 134,A -86.276,B 24.9631,C -1.4034,E1 25.0199,E2 532.594} C_DIS
LIN {X 17.4363,Y -124.1098,Z 134,A -84.9878,B 24.9631,C -1.4023,E1 25.0235,E2 531.3095} C_DIS
LIN {X 21.8539,Y -123.4083,Z 134,A -83.0438,B 24.9633,C -1.3988,E1 25.0288,E2 529.3757} C_DIS
LIN {X 24.6945,Y -122.8716,Z 134,A -81.5754,B 24.9629,C -1.4073,E1 25.0329,E2 527.889} C_DIS
LIN {X 28.6386,Y -122.0145,Z 134,A -79.6359,B 24.9626,C -1.4137,E1 25.0382,E2 525.9368} C_DIS
LIN {X 31.8339,Y -121.2186,Z 134,A -78.3882,B 24.9632,C -1.4024,E1 25.0415,E2 524.7179} C_DIS
LIN {X 35.0242,Y -120.3348,Z 134,A -76.7957,B 24.9629,C -1.4081,E1 25.0458,E2 523.1146} C_DIS
LIN {X 37.8414,Y -119.479,Z 134,A -75.6029,B 24.9632,C -1.402,E1 25.049,E2 521.9384} C_DIS
LIN {X 40.8337,Y -118.4895,Z 134,A -73.9999,B 24.9627,C -1.4119,E1 25.0533,E2 520.3149} C_DIS
LIN {X 43.6657,Y -117.4756,Z 134,A -72.5982,B 24.9625,C -1.4151,E1 25.0569,E2 518.9086} C_DIS
LIN {X 46.1658,Y -116.5177,Z 134,A -71.3925,B 24.9625,C -1.4159,E1 25.0601,E2 517.7037} C_DIS
LIN {X 49.304,Y -115.2234,Z 134,A -69.7879,B 24.9622,C -1.4209,E1 25.0642,E2 516.0911} C_DIS
LIN {X 52.4052,Y -113.8456,Z 134,A -68.4204,B 24.9625,C -1.414,E1 25.0677,E2 514.7433} C_DIS
LIN {X 54.737,Y -112.7456,Z 134,A -66.9625,B 24.9617,C -1.4301,E1 25.0714,E2 513.2512} C_DIS
LIN {X 58.0783,Y -111.0587,Z 134,A -65.4271,B 24.962,C -1.4241,E1 25.0752,E2 511.7342} C_DIS
LIN {X 61.548,Y -109.1761,Z 134,A -63.5709,B 24.9617,C -1.4299,E1 25.0797,E2 509.8696} C_DIS
LIN {X 64.9144,Y -107.2085,Z 134,A -61.7341,B 24.9614,C -1.436,E1 25.0842,E2 508.024} C_DIS
LIN {X 68.582,Y -104.901,Z 134,A -59.7258,B 24.9611,C -1.4413,E1 25.0889,E2 506.0098} C_DIS
LIN {X 71.9101,Y -102.6481,Z 134,A -57.8952,B 24.9609,C -1.4448,E1 25.0931,E2 504.1773} C_DIS
LIN {X 75.2558,Y -100.2207,Z 134,A -56.0042,B 24.9607,C -1.4489,E1 25.0974,E2 502.2833} C_DIS
LIN {X 78.8084,Y -97.4515,Z 134,A -54.0569,B 24.9607,C -1.4477,E1 25.1016,E2 500.3461} C_DIS
LIN {X 81.914,Y -94.856,Z 134,A -52.1509,B 24.9604,C -1.4548,E1 25.1057,E2 498.4306} C_DIS
LIN {X 85.115,Y -91.9953,Z 134,A -50.1466,B 24.96,C -1.4616,E1 25.1098,E2 496.4184} C_DIS
LIN {X 88.2175,Y -89.0238,Z 134,A -48.2386,B 24.9599,C -1.4636,E1 25.1136,E2 494.5138} C_DIS
LIN {X 91.0515,Y -86.1231,Z 134,A -46.3946,B 24.9596,C -1.4677,E1 25.1172,E2 492.6679} C_DIS
LIN {X 93.8079,Y -83.1122,Z 134,A -44.5403,B 24.9594,C -1.472,E1 25.1207,E2 490.8119} C_DIS
LIN {X 96.6917,Y -79.739,Z 134,A -42.5417,B 24.9592,C -1.4758,E1 25.1243,E2 488.8134} C_DIS
LIN {X 99.3061,Y -76.4591,Z 134,A -40.5912,B 24.9588,C -1.4827,E1 25.1276,E2 486.8557} C_DIS
LIN {X 101.7154,Y -73.2235,Z 134,A -38.7366,B 24.9585,C -1.4884,E1 25.1307,E2 484.9966} C_DIS
LIN {X 104.2581,Y -69.5542,Z 134,A -36.8017,B 24.9585,C -1.4887,E1 25.1337,E2 483.0707} C_DIS
LIN {X 106.3234,Y -66.3544,Z 134,A -35.0279,B 24.9581,C -1.4955,E1 25.1364,E2 481.2898} C_DIS
LIN {X 108.6326,Y -62.5029,Z 134,A -32.9559,B 24.9577,C -1.5025,E1 25.1393,E2 479.2119} C_DIS
LIN {X 110.5918,Y -58.9674,Z 134,A -31.2362,B 24.9577,C -1.5013,E1 25.1416,E2 477.5039} C_DIS
LIN {X 112.2545,Y -55.7324,Z 134,A -29.6056,B 24.9576,C -1.5047,E1 25.1437,E2 475.874} C_DIS
LIN {X 113.4249,Y -53.315,Z 134,A -28.2313,B 24.9569,C -1.5161,E1 25.1453,E2 474.4804} C_DIS
LIN {X 114.9101,Y -50.0286,Z 134,A -26.7504,B 24.9571,C -1.5125,E1 25.147,E2 473.0161} C_DIS
LIN {X 116.1325,Y -47.1213,Z 134,A -25.3282,B 24.9569,C -1.5159,E1 25.1485,E2 471.5935} C_DIS
LIN {X 117.0936,Y -44.6855,Z 134,A -23.9677,B 24.9562,C -1.5282,E1 25.1499,E2 470.2117} C_DIS
LIN {X 118.3112,Y -41.3481,Z 134,A -22.5207,B 24.9565,C -1.5241,E1 25.1512,E2 468.7824} C_DIS
LIN {X 119.3213,Y -38.3351,Z 134,A -21.1081,B 24.9563,C -1.5267,E1 25.1524,E2 467.3718} C_DIS
LIN {X 120.1918,Y -35.5128,Z 134,A -19.7237,B 24.956,C -1.5328,E1 25.1536,E2 465.9809} C_DIS
LIN {X 121.0172,Y -32.5893,Z 134,A -18.5451,B 24.9564,C -1.5263,E1 25.1544,E2 464.8244} C_DIS
LIN {X 121.7669,Y -29.6657,Z 134,A -17.0726,B 24.9558,C -1.5356,E1 25.1554,E2 463.3385} C_DIS
LIN {X 122.4417,Y -26.7446,Z 134,A -15.5927,B 24.9552,C -1.5458,E1 25.1564,E2 461.8432} C_DIS
LIN {X 123.2382,Y -22.8045,Z 134,A -13.6761,B 24.9546,C -1.5559,E1 25.1574,E2 459.914} C_DIS
LIN {X 123.8089,Y -19.4578,Z 134,A -12.2159,B 24.9546,C -1.5562,E1 25.158,E2 458.4616} C_DIS
LIN {X 124.2901,Y -16.0993,Z 134,A -10.6776,B 24.9544,C -1.5606,E1 25.1586,E2 456.9219} C_DIS
LIN {X 124.7269,Y -12.2668,Z 134,A -9.1617,B 24.9548,C -1.5535,E1 25.1591,E2 455.4318} C_DIS
LIN {X 124.9885,Y -9.2241,Z 134,A -7.6464,B 24.9542,C -1.5643,E1 25.1594,E2 453.9001} C_DIS
LIN {X 125.142,Y -6.8559,Z 134,A -6.5867,B 24.954,C -1.5665,E1 25.1596,E2 452.8414} C_DIS
LIN {X 125.2787,Y -3.5309,Z 134,A -5.0539,B 24.9537,C -1.5721,E1 25.1597,E2 451.3045} C_DIS
LIN {X 125.3282,Y -0.6113,Z 134,A -3.5915,B 24.953,C -1.5832,E1 25.1597,E2 449.8247} C_DIS
LIN {X 125.2995,Y 2.7818,Z 134,A -2.0122,B 24.9526,C -1.5897,E1 25.1597,E2 448.2394} C_DIS
LIN {X 125.1338,Y 7.0147,Z 134,A -0.2339,B 24.9528,C -1.5878,E1 25.1595,E2 446.4762} C_DIS
LIN {X 124.8958,Y 10.4047,Z 134,A 1.2599,B 24.9526,C -1.5897,E1 25.1592,E2 444.9867} C_DIS
LIN {X 124.6742,Y 12.8024,Z 134,A 2.5124,B 24.952,C -1.6012,E1 25.1588,E2 443.7146} C_DIS
LIN {X 124.2796,Y 16.1788,Z 134,A 3.9105,B 24.9521,C -1.5981,E1 25.1583,E2 442.332} C_DIS
LIN {X 123.8979,Y 18.8826,Z 134,A 5.2585,B 24.9516,C -1.6073,E1 25.1578,E2 440.9703} C_DIS
LIN {X 123.4188,Y 21.7953,Z 134,A 6.4936,B 24.9516,C -1.6057,E1 25.1572,E2 439.7462} C_DIS
LIN {X 122.8716,Y 24.6945,Z 134,A 7.949,B 24.9511,C -1.6155,E1 25.1564,E2 438.2761} C_DIS
LIN {X 122.0046,Y 28.6797,Z 134,A 9.8687,B 24.9506,C -1.6243,E1 25.1552,E2 436.3471} C_DIS
LIN {X 121.1916,Y 31.9352,Z 134,A 11.1105,B 24.9512,C -1.6139,E1 25.1544,E2 435.1368} C_DIS
LIN {X 120.4925,Y 34.4857,Z 134,A 12.5889,B 24.9501,C -1.6316,E1 25.1533,E2 433.6251} C_DIS
LIN {X 119.479,Y 37.8414,Z 134,A 13.8794,B 24.9508,C -1.6204,E1 25.1522,E2 432.3684} C_DIS
LIN {X 118.5328,Y 40.7089,Z 134,A 15.4877,B 24.9498,C -1.6364,E1 25.1508,E2 430.7315} C_DIS
LIN {X 117.4756,Y 43.6657,Z 134,A 16.8635,B 24.9498,C -1.6376,E1 25.1495,E2 429.3605} C_DIS
LIN {X 116.5011,Y 46.207,Z 134,A 18.0725,B 24.9496,C -1.6395,E1 25.1482,E2 428.1539} C_DIS
LIN {X 115.2031,Y 49.3509,Z 134,A 19.6824,B 24.9492,C -1.6469,E1 25.1465,E2 426.5353} C_DIS
LIN {X 113.8888,Y 52.3119,Z 134,A 21.0492,B 24.9492,C -1.6453,E1 25.1449,E2 425.1796} C_DIS
LIN {X 112.7456,Y 54.737,Z 134,A 22.4964,B 24.9483,C -1.6602,E1 25.1431,E2 423.705} C_DIS
LIN {X 111.3213,Y 57.5782,Z 134,A 23.9367,B 24.9481,C -1.6637,E1 25.1413,E2 422.2642} C_DIS
LIN {X 109.1761,Y 61.548,Z 134,A 25.8765,B 24.9481,C -1.6631,E1 25.1387,E2 420.336} C_DIS
LIN {X 107.3297,Y 64.714,Z 134,A 27.6192,B 24.9477,C -1.6711,E1 25.1362,E2 418.5834} C_DIS
LIN {X 104.9491,Y 68.5078,Z 134,A 29.5579,B 24.9477,C -1.6709,E1 25.1333,E2 416.6548} C_DIS
LIN {X 102.7847,Y 71.7138,Z 134,A 31.3754,B 24.9472,C -1.678,E1 25.1304,E2 414.8295} C_DIS
LIN {X 100.2791,Y 75.1784,Z 134,A 33.3921,B 24.9467,C -1.6861,E1 25.1271,E2 412.8034} C_DIS
LIN {X 97.8084,Y 78.3659,Z 134,A 35.2081,B 24.9465,C -1.6892,E1 25.1239,E2 410.9885} C_DIS
LIN {X 95.2124,Y 81.5002,Z 134,A 37.0716,B 24.9462,C -1.6938,E1 25.1206,E2 409.1228} C_DIS
LIN {X 92.3809,Y 84.6955,Z 134,A 38.9849,B 24.9461,C -1.6963,E1 25.117,E2 407.212} C_DIS
LIN {X 89.3624,Y 87.8744,Z 134,A 40.9747,B 24.9458,C -1.7,E1 25.1131,E2 405.222} C_DIS
LIN {X 86.2984,Y 90.8861,Z 134,A 42.9616,B 24.9455,C -1.7054,E1 25.1091,E2 403.2308} C_DIS
LIN {X 83.1336,Y 93.789,Z 134,A 44.9007,B 24.9453,C -1.7082,E1 25.1051,E2 401.2929} C_DIS
LIN {X 79.6523,Y 96.7635,Z 134,A 47.003,B 24.945,C -1.7127,E1 25.1006,E2 399.188} C_DIS
LIN {X 76.2684,Y 99.4519,Z 134,A 48.9407,B 24.945,C -1.7145,E1 25.0963,E2 397.2532} C_DIS
LIN {X 72.7628,Y 102.0448,Z 134,A 50.9204,B 24.9447,C -1.7173,E1 25.0919,E2 395.2739} C_DIS
LIN {X 69.2525,Y 104.4595,Z 134,A 52.8905,B 24.9445,C -1.7216,E1 25.0873,E2 393.3} C_DIS
LIN {X 65.6698,Y 106.7476,Z 134,A 54.7993,B 24.9444,C -1.723,E1 25.0828,E2 391.3942} C_DIS
LIN {X 61.7962,Y 109.0362,Z 134,A 56.8808,B 24.9441,C -1.7272,E1 25.0777,E2 389.3089} C_DIS
LIN {X 58.5039,Y 110.8352,Z 134,A 58.3069,B 24.9449,C -1.7152,E1 25.0743,E2 387.9153} C_DIS
LIN {X 55.7324,Y 112.2545,Z 134,A 59.8742,B 24.9443,C -1.7242,E1 25.0704,E2 386.3311} C_DIS
LIN {X 53.315,Y 113.4249,Z 134,A 61.2573,B 24.9437,C -1.7334,E1 25.0668,E2 384.9298} C_DIS
LIN {X 50.0286,Y 114.9101,Z 134,A 62.7407,B 24.9441,C -1.7271,E1 25.0631,E2 383.4649} C_DIS
LIN {X 47.0606,Y 116.157,Z 134,A 64.1808,B 24.9441,C -1.7271,E1 25.0594,E2 382.0281} C_DIS
LIN {X 44.6855,Y 117.0936,Z 134,A 65.5334,B 24.9434,C -1.7374,E1 25.0558,E2 380.6541} C_DIS
LIN {X 41.3481,Y 118.3112,Z 134,A 66.9898,B 24.9439,C -1.7306,E1 25.052,E2 379.2167} C_DIS
LIN {X 38.5543,Y 119.2513,Z 134,A 68.371,B 24.9437,C -1.7334,E1 25.0483,E2 377.8316} C_DIS
LIN {X 35.5128,Y 120.1918,Z 134,A 69.8016,B 24.9437,C -1.7334,E1 25.0445,E2 376.4038} C_DIS
LIN {X 32.5893,Y 121.0172,Z 134,A 70.9856,B 24.9443,C -1.7242,E1 25.0414,E2 375.2431} C_DIS
LIN {X 29.5448,Y 121.796,Z 134,A 72.4971,B 24.944,C -1.7288,E1 25.0373,E2 373.7232} C_DIS
LIN {X 26.7446,Y 122.4417,Z 134,A 73.9625,B 24.9435,C -1.7368,E1 25.0333,E2 372.2406} C_DIS
LIN {X 22.7835,Y 123.242,Z 134,A 75.886,B 24.9432,C -1.7413,E1 25.028,E2 370.3088} C_DIS
LIN {X 19.3177,Y 123.8306,Z 134,A 77.2422,B 24.9439,C -1.7297,E1 25.0243,E2 368.9815} C_DIS
LIN {X 16.5782,Y 124.2273,Z 134,A 78.6892,B 24.9433,C -1.7388,E1 25.0202,E2 367.5141} C_DIS
LIN {X 13.6816,Y 124.5796,Z 134,A 79.9465,B 24.9436,C -1.7353,E1 25.0168,E2 366.266} C_DIS
LIN {X 9.2048,Y 124.9899,Z 134,A 81.9519,B 24.9437,C -1.7331,E1 25.0112,E2 364.267} C_DIS
LIN {X 6.7783,Y 125.1459,Z 134,A 83.023,B 24.9438,C -1.7311,E1 25.0082,E2 363.2009} C_DIS
LIN {X 3.5364,Y 125.2785,Z 134,A 84.575,B 24.9436,C -1.7343,E1 25.0039,E2 361.6418} C_DIS
LIN {X 0.4124,Y 125.3281,Z 134,A 86.0594,B 24.9435,C -1.7368,E1 24.9997,E2 360.1517} C_DIS
LIN {X -3.3987,Y 125.2823,Z 134,A 87.7315,B 24.9437,C -1.733,E1 24.9951,E2 358.4885} C_DIS
LIN {X -6.0066,Y 125.1847,Z 134,A 88.84,B 24.944,C -1.7285,E1 24.992,E2 357.3903} C_DIS
LIN {X -8.4145,Y 125.0476,Z 134,A 90.2362,B 24.9431,C -1.7421,E1 24.988,E2 355.9615} C_DIS
LIN {X -12.7469,Y 124.6802,Z 134,A 92.1806,B 24.9433,C -1.739,E1 24.9827,E2 354.0233} C_DIS
LIN {X -16.1068,Y 124.2891,Z 134,A 93.5825,B 24.9438,C -1.7313,E1 24.9788,E2 352.6389} C_DIS
LIN {X -19.9006,Y 123.7403,Z 134,A 95.5162,B 24.9433,C -1.7386,E1 24.9734,E2 350.6861} C_DIS
LIN {X -23.1673,Y 123.1689,Z 134,A 96.9149,B 24.9438,C -1.7319,E1 24.9696,E2 349.3018} C_DIS
LIN {X -26.3633,Y 122.524,Z 134,A 98.3756,B 24.944,C -1.7292,E1 24.9656,E2 347.8458} C_DIS
LIN {X -30.5343,Y 121.552,Z 134,A 100.295,B 24.9442,C -1.7255,E1 24.9604,E2 345.9325} C_DIS
LIN {X -33.1023,Y 120.8794,Z 134,A 101.5383,B 24.9442,C -1.7256,E1 24.9571,E2 344.6871} C_DIS
LIN {X -36.3806,Y 119.9319,Z 134,A 103.1385,B 24.9442,C -1.7258,E1 24.9528,E2 343.0839} C_DIS
LIN {X -38.867,Y 119.1514,Z 134,A 104.4915,B 24.9438,C -1.7319,E1 24.9492,E2 341.7139} C_DIS
Enddeposition()
END
